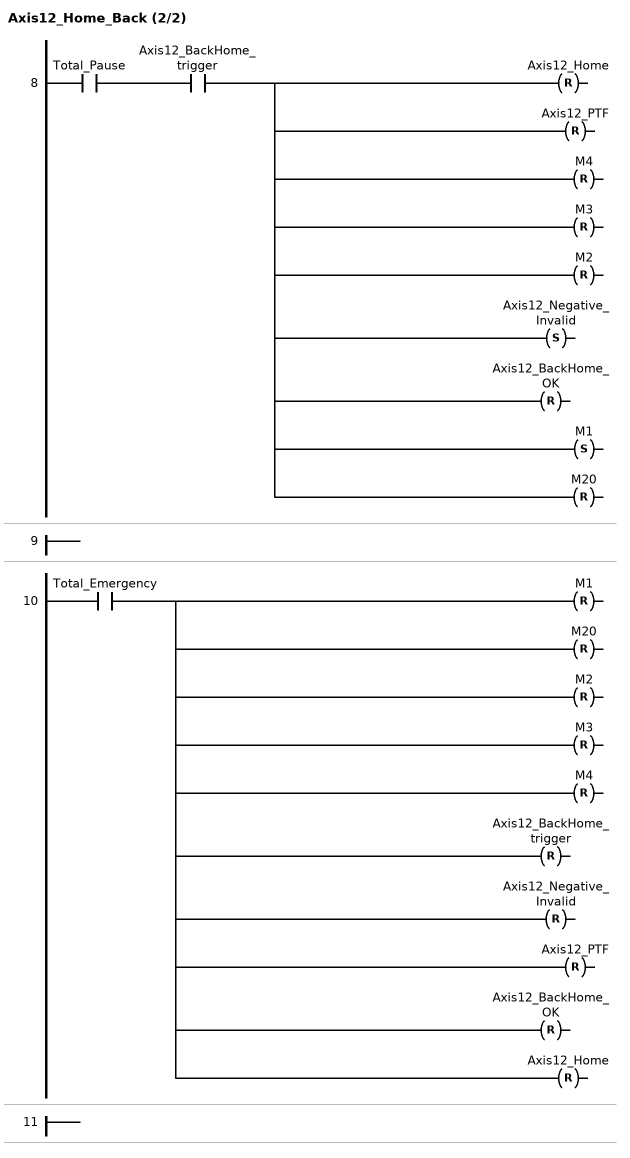
[picture p96: Axis12_Home_Back (LD)]
_LD_ (* Ladder Diagram *)
NETWORK 1
	[Axis12_BackHome_trigger] - UP1:R_TRIG(CLK: *) --- (S M1) (S Axis12_Negative_Invalid)
NETWORK 2
	[M1] - [/Total_Pause] --- (S Axis12_PTF) (S M2) (R M1)
NETWORK 3
	[M2] - [Axis12_Negative_Limit] --- (S Axis12_Halt) (S M20) (R M2) (R Axis12_PTF)
NETWORK 4
	[M20] - [Axis12_Halt_Function.Done] - T1:TON(IN: *, PT: T#1MS) --- (R Axis12_Halt) (S M3) (R M20)
NETWORK 5
	[M3] - [/Total_Pause] --- (S M4) (S Axis12_Home)
NETWORK 6
	[M4] - [Axis12_Negative_Limit] - DOWN1:F_TRIG(CLK: *) --- (R Axis12_Negative_Invalid)
NETWORK 7
	[M4] - [Axis12_Home_Function.Done] --- (S Axis12_BackHome_OK) (R Axis12_Home) (R Axis12_BackHome_trigger) (R M4) (R M3)
NETWORK 8
	[Total_Pause] - [Axis12_BackHome_trigger] --- (R Axis12_Home) (R Axis12_PTF) (R M4) (R M3) (R M2) (S Axis12_Negative_Invalid) (R Axis12_BackHome_OK) (S M1) (R M20)
NETWORK 9
	*
NETWORK 10
	[Total_Emergency] --- (R M1) (R M20) (R M2) (R M3) (R M4) (R Axis12_BackHome_trigger) (R Axis12_Negative_Invalid) (R Axis12_PTF) (R Axis12_BackHome_OK) (R Axis12_Home)
NETWORK 11
	*
_END_LD_
(* the same logic as Structured Text *)
(* Network 1 *)
UP1(CLK := Axis12_BackHome_trigger);
IF UP1.Q THEN M1 := TRUE; Axis12_Negative_Invalid := TRUE; END_IF;
(* Network 2 *)
_p1 := M1 AND NOT Total_Pause;
IF _p1 THEN Axis12_PTF := TRUE; M2 := TRUE; M1 := FALSE; END_IF;
(* Network 3 *)
_p2 := M2 AND Axis12_Negative_Limit;
IF _p2 THEN Axis12_Halt := TRUE; M20 := TRUE; M2 := FALSE; Axis12_PTF := FALSE; END_IF;
(* Network 4 *)
T1(IN := M20 AND Axis12_Halt_Function.Done, PT := T#1MS);
IF T1.Q THEN Axis12_Halt := FALSE; M3 := TRUE; M20 := FALSE; END_IF;
(* Network 5 *)
IF M3 AND NOT Total_Pause THEN M4 := TRUE; Axis12_Home := TRUE; END_IF;
(* Network 6 *)
DOWN1(CLK := M4 AND Axis12_Negative_Limit);
IF DOWN1.Q THEN Axis12_Negative_Invalid := FALSE; END_IF;
(* Network 7 *)
_p3 := M4 AND Axis12_Home_Function.Done;
IF _p3 THEN Axis12_BackHome_OK := TRUE; Axis12_Home := FALSE; Axis12_BackHome_trigger := FALSE; M4 := FALSE; M3 := FALSE; END_IF;
(* Network 8 *)
IF Total_Pause AND Axis12_BackHome_trigger THEN Axis12_Home := FALSE; Axis12_PTF := FALSE; M4 := FALSE; M3 := FALSE; M2 := FALSE; Axis12_Negative_Invalid := TRUE; Axis12_BackHome_OK := FALSE; M1 := TRUE; M20 := FALSE; END_IF;
(* Network 9 *)
(* Network 10 *)
IF Total_Emergency THEN M1 := FALSE; M20 := FALSE; M2 := FALSE; M3 := FALSE; M4 := FALSE; Axis12_BackHome_trigger := FALSE; Axis12_Negative_Invalid := FALSE; Axis12_PTF := FALSE; Axis12_BackHome_OK := FALSE; Axis12_Home := FALSE; END_IF;
(* Network 11 *)
END_PROGRAM

(* POU Other_Folder/Akam_Stop_Message/Initialization_Folder/IniRun, ST *)
PROGRAM IniRun
VAR
	step: INT;
	bak_step:INT;
	rt_hold: R_TRIG;
	M1: BOOL;

	T1: TON;
	T2:TON;


END_VAR

VAR_INPUT
	bstart1: BOOL;
	bhold1: BOOL;
	breset1: BOOL;

END_VAR
(*数据保存*)
IF Save_Button THEN
Save_Par(NETID:='',port:=801,start:=TRUE,tmout:=T#1s);
END_IF
IF NOT Save_Par.BUSY  THEN
Save_Button:=FALSE;
Save_Par(NETID:='',port:=801,start:=FALSE,tmout:=T#1s);
END_IF


(*当出现回原点没有时，需要初始化*)
IF NOT Axis1_BackHome_OK OR NOT  Axis2_BackHome_OK OR NOT Axis3_BackHome_OK OR NOT Axis4_BackHome_OK OR NOT Axis5_BackHome_OK
	OR NOT Axis6_BackHome_OK OR NOT Axis7_BackHome_OK OR NOT Axis8_BackHome_OK OR NOT Axis9_BackHome_OK OR NOT Axis10_BackHome_OK OR NOT Axis11_BackHome_OK  THEN
;(*判断是否需要回原点----------------------------------------------------*)
END_IF
(*---------------------------------------------------------------------------初始化开始流程---------------------------------------------------------------------------------*)
CASE step OF
0:
Need_Ini:=TRUE;(*此时寻妖初始化*)
(*进入初始化流程*)
step:=10;

10:(*判断是否需要初始化*)
IF Need_Ini AND NOT Total_Axis_Error AND NOT Debug_Model   THEN (*当需要初始化的时候，复位所有原点ok信号*)
	Axis1_BackHome_OK:=FALSE;
Axis2_BackHome_OK:=FALSE;
Axis3_BackHome_OK:=FALSE;
Axis4_BackHome_OK:=FALSE;
Axis5_BackHome_OK:=FALSE;
Axis6_BackHome_OK:=FALSE;
Axis7_BackHome_OK:=FALSE;
Axis8_BackHome_OK:=FALSE;
Axis9_BackHome_OK:=FALSE;
Axis10_BackHome_OK:=FALSE;
Axis11_BackHome_OK:=FALSE;
step:=20;
END_IF

20:(*等待复位按钮操作，复位报警等状态*)
IF X4_6 AND Need_Ini THEN
	IF Total_Axis_Error THEN
	M1:=TRUE;(*no use*)(*上位机提示电机报警问题，需要初始化*)
	END_IF
	IF NOT Total_Axis_Error THEN
	step:=30;
	END_IF
END_IF;

30:(*启动按下的处理开始进入初始化过中。。。。。。*)
IF X4_4 AND NOT Total_Axis_Error AND NOT Debug_Model THEN
Need_Ini:=FALSE;
IsIniing:=TRUE;(*初始化中ing*)
M101:=TRUE;(*初始化中，速度为中速*)
Axis1_Poweron:=TRUE;
Axis2_Poweron:=TRUE;
Axis3_Poweron:=TRUE;
Axis4_Poweron:=TRUE;
Axis5_Poweron:=TRUE;
Axis6_Poweron:=TRUE;
Axis7_Poweron:=TRUE;
Axis8_Poweron:=TRUE;
Axis9_Poweron:=TRUE;
Axis10_Poweron:=TRUE;
Axis11_Poweron:=TRUE;
step:=39;
END_IF

39:
(*滑台气缸上下，如果在同一高度，则说明不存在重叠部分，可复位气缸*)
IF (X4_11 AND X4_13) OR (X4_12 AND X4_14)  AND X2_6 THEN
Y1_6:=FALSE;
Y1_7:=FALSE;
step:=40;
ELSE
step:=40;
END_IF


40:(*气缸复位状态保留*)

Y0_2:=FALSE;
Y0_5:=FALSE;
Y0_14:=FALSE;
y0_1:=TRUE;
Y0_12:=FALSE;



(******************** AND  *****************************)

Y0_7:=FALSE;(*左上下气缸*)
Y0_9:=FALSE;(*滚压气缸复位*)
Y1_1:=FALSE;(*右上下气缸*)
Y0_4:=FALSE;
Y1_3:=FALSE;
IF X2_13 AND X3_3 AND X3_11 THEN
	step:=50;(*初步气缸复位*)
END_IF

50:
Y0_6:=FALSE;(*左平移气缸复位*)
Y0_11:=FALSE;(*滚压部分下压气缸复位*)
Y0_16:=FALSE;(*右平移气缸复位*)
T1(IN:=TRUE , PT:=t#1s , Q=> , ET=> );
IF T1.Q AND X2_11 AND X3_9 THEN
T1(IN:=FALSE , PT:=t#1s , Q=> , ET=> );
step:=60;(*无感气缸*)
END_IF

60:(*复位滚压气缸部分气缸，推入气缸，和翻转气缸*)
Y0_10:=FALSE;
IF X3_1 THEN
step:=70;
END_IF

70:(*翻转气缸复位*)
Y0_13:=FALSE;
IF X3_5 THEN
step:=80;
END_IF

80:(*上电延时*)
T2(IN:=TRUE , PT:=t#1s , Q=> , ET=> );
IF T2.Q  AND NOT Total_Pause THEN
T2(IN:=FALSE , PT:=t#1s , Q=> , ET=> );
step:=90;
END_IF

90:
home_backing:=TRUE;
IF NOT Axis3_BackHome_OK OR NOT Axis6_BackHome_OK OR NOT Axis7_BackHome_OK OR NOT Axis8_BackHome_OK OR NOT Axis9_BackHome_OK THEN
step:=100;
ELSE
step:=110;(*当喂料都已经回过原点，则不需要回原点*)
END_IF


100:(*判断是否都需要回原点*)(*喂料部分回原点*)
Axis3_BackHome_trigger:=TRUE;(**)
Axis6_BackHome_trigger:=TRUE;(**)
Axis7_BackHome_trigger:=TRUE;(**)
Axis8_BackHome_trigger:=TRUE;(**)
Axis9_BackHome_trigger:=TRUE;
IF Axis3_BackHome_OK AND Axis6_BackHome_OK AND Axis7_BackHome_OK AND Axis8_BackHome_OK AND Axis9_BackHome_OK  THEN
Axis3_BackHome_trigger:=FALSE;(**)
Axis6_BackHome_trigger:=FALSE;(**)
Axis7_BackHome_trigger:=FALSE;(**)
Axis8_BackHome_trigger:=FALSE;(**)
Axis9_BackHome_trigger:=FALSE;
step:=101;
END_IF

101:(*升降回到初始位置*)
D3:=D300;(*进料初始位置，在下面*)
D6:=D600;(*上升初始位置，在下面*)
D7:=D700;(*下降初始位置，在下面*)
D8:=D800;(*上升初始位置，在下面*)
D9:=D900;(*下降初始位置，在下面*)
Axis3_MoveAbsolute:=TRUE;
Axis6_MoveAbsolute:=TRUE;
Axis7_MoveAbsolute:=TRUE;
Axis8_MoveAbsolute:=TRUE;
Axis9_MoveAbsolute:=TRUE;
IF Axis3_Abs_Function.Done AND Axis6_Abs_Function.Done AND Axis7_Abs_Function.Done AND Axis8_Abs_Function.Done AND Axis9_Abs_Function.Done  THEN
Axis3_MoveAbsolute:=FALSE;
Axis6_MoveAbsolute:=FALSE;
Axis7_MoveAbsolute:=FALSE;
Axis8_MoveAbsolute:=FALSE;
Axis9_MoveAbsolute:=FALSE;
step:=102;  (*初始都在下面*)
END_IF

102:(*Z轴撕膜电机回原*)
Axis5_BackHome_trigger:=TRUE;
IF Axis5_BackHome_OK THEN
Axis5_BackHome_trigger:=FALSE;
step:=103;
END_IF

103:
D5:=A5_W0;(*Z轴回到初始位置*)
Axis5_MoveAbsolute:=TRUE;
IF Axis5_Abs_Function.Done THEN
Axis5_MoveAbsolute:=FALSE;
step:=110;
END_IF

110:(*其余轴回原点*)
Axis1_BackHome_trigger:=TRUE;
Axis11_BackHome_trigger:=TRUE;
Axis2_BackHome_trigger:=TRUE;
Axis4_BackHome_trigger:=TRUE;
Axis10_BackHome_trigger:=TRUE;
IF Axis1_BackHome_OK AND Axis2_BackHome_OK AND Axis4_BackHome_OK  AND Axis10_BackHome_OK AND Axis11_BackHome_OK  THEN
Axis1_BackHome_trigger:=FALSE;
Axis2_BackHome_trigger:=FALSE;
Axis4_BackHome_trigger:=FALSE;
Axis10_BackHome_trigger:=FALSE;
Axis11_BackHome_trigger:=FALSE;
step:=120;
END_IF

120:(*移载等轴的回到初始位置*)
D1:=A1_W0;
D1_1:=A11_W0+250;(*为了保证回原点之后，滑台1气缸在下面，滑台2气缸在上面，则需要，错开初始位置*)
D2:=A2_W0;
D4:=A4_W0;
D10:=A10_W0;
Axis1_MoveAbsolute:=TRUE;
Axis2_MoveAbsolute:=TRUE;
Axis4_MoveAbsolute:=TRUE;
Axis10_MoveAbsolute:=TRUE;
Axis11_MoveAbsolute:=TRUE;
IF Axis1_Abs_Function.Done AND Axis2_Abs_Function.Done AND Axis4_Abs_Function.Done  AND Axis10_Abs_Function.Done AND Axis11_Abs_Function.Done  THEN
Axis1_MoveAbsolute:=FALSE;
Axis2_MoveAbsolute:=FALSE;
Axis4_MoveAbsolute:=FALSE;
Axis10_MoveAbsolute:=FALSE;
Axis11_MoveAbsolute:=FALSE;
home_backing:=FALSE;
Y1_6:=FALSE;(*最终保证，滑台1在上面，滑台2气缸在下面*)
Y1_7:=FALSE;
step:=121;
END_IF


121:
IF  X4_11 AND X4_14 THEN(*最终结果，传感器检测*)
step:=122;
END_IF

122:
D1_1:=A11_W0;
Axis11_MoveAbsolute:=TRUE;
IF  Axis11_Abs_Function.Done THEN
Axis11_MoveAbsolute:=FALSE;
step:=130;
END_IF


130:(*其余需要初始化的状态*)

IsIniing:=FALSE;
Model_Choose:=TRUE;(*模式选择*)
step:=140;

140:
(*模式选选择，直接按钮，启动程序，当选上位机选择调试模式，同时按下启动按钮，则进入调试模式*)
IF NOT Debug_Model AND X4_4 THEN
	Model_Choose:=FALSE;(*模式选择*)
Product_Film_Handel_Run:=TRUE;
Left_Translation_Run_1:=TRUE;
Left_Translation_Run_2:=TRUE;
Right_Translation_Run:=TRUE;
Rolling_Part_Run:=TRUE;
Right_Carry_Run:=TRUE;
Left_Carry_Run:=TRUE;
Liftin_Feed_1_Run:=TRUE;
Liftin_Feed_Left_1_Run:=TRUE;
Liftin_Feed_Left_2_Run:=TRUE;
Liftin_Feed_Right_1_Run:=TRUE;
Liftin_Feed_Right_2_Run:=TRUE;
M102:=TRUE;
Debug_Model:=FALSE;
Positive2_Safe:=TRUE;
	Positive3_Safe:=TRUE;
	Positive_Wait_Safe:=TRUE;
runing:=TRUE;
	step:=150;
END_IF
IF Debug_Model AND X4_4 THEN
	M100:=TRUE;(*调试模式下低速*)
	Model_Choose:=FALSE;(*模式选择*)
	Axis1_debug_trigger:=TRUE;
Axis1_debug_trigger:=TRUE;
Axis2_debug_trigger:=TRUE;
Axis3_debug_trigger:=TRUE;
Axis4_debug_trigger:=TRUE;
Axis5_debug_trigger:=TRUE;
Axis6_debug_trigger:=TRUE;
Axis7_debug_trigger:=TRUE;
Axis8_debug_trigger:=TRUE;
Axis9_debug_trigger:=TRUE;
Axis10_debug_trigger:=TRUE;
Axis11_debug_trigger:=TRUE;
(*其余调试模式*)
 step:=160;
END_IF

150:(*运行模式下的死循环*)
;


160:
(*调试模式下的死循环，等待调试模式借宿，重新开始初始化*)
IF NOT Debug_Model THEN
Need_Ini:=TRUE;
 	    bak_step:=0;
	step:=0;
END_IF



300:(*外部输入启动*)
    IF bstart1   AND NOT Total_Axis_Error AND NOT total_pausestatus THEN
	step:=bak_step;
END_IF;
END_CASE;



(*触发暂停的外部输入*)
rt_hold(CLK:=( Total_Axis_Error OR  bhold1) , Q=> ); (*暂停状态*)
IF step<>0 AND step<>300   AND  rt_hold.Q THEN
     bak_step:=step;
     step:=300;
END_IF

(*急停处理*)
IF Total_Emergency THEN
debug_FLIG:=FALSE;
M100:=FALSE;
M101:=FALSE;
M102:=FALSE;
IsIniing:=FALSE;
runing:=FALSE;
home_backing:=FALSE;
Model_Choose:=FALSE;(*模式选择*)


Debug_Model:=FALSE;
Positive2_Safe:=FALSE;
Positive3_Safe:=FALSE;
Positive_Wait_Safe:=FALSE;


bak_step:=0;
step:=0;
END_IF


(*与debug1中的梯形图一起使用，当不在应该调试模式下的时候，按下调试按钮，自动复位--------详见------debug1----------*)
IF step<>160 AND step<>140 AND step<>300  THEN
debug_FLIG:=FALSE;
ELSE
debug_FLIG:=TRUE;
END_IF
END_PROGRAM

(* POU old/Old_Tray_Pro/Liftin_Feed_Right_1, ST *)
PROGRAM Liftin_Feed_Right_1
VAR

	step: INT;
	bak_step:INT;
	rt_hold: R_TRIG;
	UP1: R_TRIG;
	T1: TON;
	T2:TON;

END_VAR

VAR_INPUT
	bstart1: BOOL;
	bhold1: BOOL;
	breset1: BOOL;

END_VAR
UP1(CLK:=Liftin_Feed_Right_1_Run , Q=> );

CASE step OF
0:
 IF UP1.Q THEN
step:=10;
END_IF


10:(*上升运行*)
Axis8_PTF_2:=TRUE;
IF X2_4 AND  X1_3 THEN(*碰到光纤，同时没有碰到极限，此时上料ok*)
Axis8_PTF_2:=FALSE;
Feed_3_Finish:=TRUE;
Axis8_Halt:=TRUE;
step:=20;
END_IF
IF NOT X1_3 THEN(*碰到极限，此时表示料空*)
Axis8_PTF_2:=FALSE;
Axis8_Halt:=TRUE;
step:=50;
END_IF

20:
Axis8_Halt:=FALSE;
(*表示上料成功,等待取完信号*)
IF Get_Robort3_Tray_Full THEN
Feed_3_Finish:=FALSE;
Get_Robort3_Tray_Full:=FALSE;(*放满信号，给出，等待移动*)
Right_Can_Move:=TRUE;
step:=30;
END_IF


30:(*等待平移完成，才可以上升*)
IF Right_Move_Finish THEN
Right_Move_Finish:=FALSE;
step:=10;
END_IF


50:(*碰到极限，此时料取完,回到初始位置*)
Axis8_Halt:=FALSE;
D8:=D800;
Axis8_MoveAbsolute:=TRUE;
IF Axis8_Abs_Function.Done THEN
Axis8_MoveAbsolute:=FALSE;
Feed_Right_None_Alam:=TRUE;(*不暂停，只提示*)
step:=60;
END_IF

60:(*回到初始位置，提示料空*)
IF Right_UP_Button AND NOT Total_Pause THEN
Right_UP_Button:=FALSE;
Feed_Right_None_Alam:=FALSE;(*不暂停，只提示*)
step:=10;
END_IF

300:
    IF bstart1   AND NOT Total_Axis_Error AND NOT total_pausestatus THEN
	step:=bak_step;
END_IF;
END_CASE


rt_hold(CLK:=( Total_Axis_Error OR  bhold1) , Q=> ); (*暂停状态*)
IF step<>0 AND step<>300   AND  rt_hold.Q THEN
     bak_step:=step;
     step:=300;
END_IF


IF Right_UP_Button THEN
Right_UP_Button:=FALSE;
END_IF

IF Total_Emergency THEN
Liftin_Feed_Right_1_Run:=FALSE;
Feed_Right_None_Alam:=FALSE;
Feed_3_Finish:=FALSE;


bak_step:=0;
step:=0;
END_IF


(*随时可以不做料的操作*)
IF Feed_Right_Button1 AND step=20 AND NOT Total_Pause THEN
Feed_Right_Button1:=FALSE;
Feed_3_Finish:=FALSE;
step:=50;
ELSE
Feed_Right_Button1:=FALSE;
END_IF
END_PROGRAM

(* POU old/Old_Tray_Pro/Liftin_Feed_Right_2, ST *)
PROGRAM Liftin_Feed_Right_2
VAR

	step: INT;
	bak_step:INT;
	rt_hold: R_TRIG;
	UP1: R_TRIG;
	DOWN1: F_TRIG;

	T1: TON;
	T2:TON;

END_VAR

VAR_INPUT
	bstart1: BOOL;
	bhold1: BOOL;
	breset1: BOOL;

END_VAR
(*左下降，初始化，回原点到初始位置，，，启动之后，先往上走，到初始位置(第一次回原点使用)  ，接收到送料完成可下降信号，则
开始下降，等现将结束，告知，可放料*)

UP1(CLK:=Liftin_Feed_Right_2_Run , Q=> );

CASE step OF
0:
 IF UP1.Q THEN
step:=1;
END_IF

1:
(*初始化之后位置在下面的初始位置*)
Axis9_PTF_2:=TRUE;
IF X2_5 AND X1_6 THEN
Axis9_PTF_2:=FALSE;
Axis9_Halt:=TRUE;
step:=20;
END_IF
IF NOT X1_6 THEN
Axis9_PTF_2:=FALSE;
Axis9_Halt:=TRUE;
step:=60;(*撞到极限，此时需要回到上面的初始位置*)
END_IF

10:
(*初始化的时候写，回原点之后，向上跑知道碰到光纤，或者极限的时候，到极限回到初始位置，碰到光纤，停止，翻转到极限停止位置*)

(*到初始位置，等待放料，当光纤感应到，同时，接收到，可下降信号的时候，开始下降，当感应不到光纤，则停止*)
IF you_ke_jiang AND X2_5 THEN
you_ke_jiang:=FALSE;
	step:=20;
END_IF

20:
Axis9_Halt:=FALSE;
(*接收到可降信号，开始下降，到传感器下降沿停止下降，等待*)
Axis9_PTF:=TRUE;
DOWN1(CLK:=X2_5 , Q=> );
IF DOWN1.Q AND NOT  X1_7 THEN
Axis9_PTF:=FALSE;
you_down_Finish:=TRUE;
Axis9_Halt:=TRUE;
step:=30;
END_IF
IF  X1_7 THEN(*碰到极限，此时表示料空*)
Axis9_PTF:=FALSE;
Axis9_Halt:=TRUE;
step:=400;
END_IF

30:(*停止，给出下降完成信号，等待放料循环*)
Axis9_Halt:=FALSE;
step:=10;

400:(*碰到原点，此时，回到下初始位置，给出料满提示*)
Axis9_Halt:=FALSE;
D9:=D900;
Axis9_MoveAbsolute:=TRUE;
IF Axis9_Abs_Function.Done THEN
Axis9_MoveAbsolute:=FALSE;
Feed_Right_None_Alam:=TRUE;(*不暂停，只提示*)
step:=50;
END_IF

50:(*碰到下极限，给出缺料提示*)
Axis9_Halt:=FALSE;
IF Right_Down_Button AND NOT Total_Pause THEN
	Right_Down_Button:=FALSE;
Feed_Right_Full_Alam:=FALSE;
	step:=1;(*确认拿走料之后，运动到初始位置*)
END_IF

60:(*回到初始位置*)
Axis9_Halt:=FALSE;
D9:=D910;
Axis9_MoveAbsolute:=TRUE;
IF Axis9_Abs_Function.Done THEN
Axis9_MoveAbsolute:=FALSE;
you_down_Finish:=TRUE;(*左下降完成信号*)
step:=10;
END_IF

300:
    IF bstart1   AND NOT Total_Axis_Error AND NOT total_pausestatus THEN
	step:=bak_step;
END_IF;
END_CASE


rt_hold(CLK:=( Total_Axis_Error OR  bhold1) , Q=> ); (*暂停状态*)
IF step<>0 AND step<>300   AND  rt_hold.Q THEN
     bak_step:=step;
     step:=300;
END_IF


IF Total_Emergency THEN
Liftin_Feed_Right_2_Run:=FALSE;
you_down_Finish:=FALSE;
Feed_Right_Full_Alam:=FALSE;


bak_step:=0;
step:=0;
END_IF


(*随时可以不做料的操作*)
IF Feed_Right_Button2 AND step=10 AND NOT Total_Pause THEN
Feed_Right_Button2:=FALSE;
you_down_Finish:=FALSE;
step:=400;
ELSE
Feed_Right_Button2:=FALSE;
END_IF
END_PROGRAM

(* POU Test_Part_pro/New_Table_3, ST *)
PROGRAM New_Table_3
VAR
	step: INT;
	bak_step:INT;
	rt_hold: R_TRIG;
	UP1: R_TRIG;
	Run_Time:BOOL;
	T1:TON;
	Run_Time_Lreal: TIME;




	T2: TON;
	T3: TON;
END_VAR

VAR_INPUT
	bstart1: BOOL;
	bhold1: BOOL;
	breset1: BOOL;

END_VAR
UP1(CLK:=Left_Translation_Run_2 , Q=> );

CASE step OF
0:
 IF UP1.Q THEN
step:=10;
END_IF

10:
D1_1:=A11_W1;(*左等待放料工位*)
Axis11_MoveAbsolute:=TRUE;
IF Axis11_Abs_Function.Done THEN
Axis11_MoveAbsolute:=FALSE;
step:=20;
END_IF;

20:(*到下初始位置------寻味位置1是否安全*)
IF Positive1_Safe THEN
	Positive1_Safe:=FALSE;
	Y1_7:=TRUE;
step:=30;
END_IF

30:
IF X4_13 THEN
	Positive4_Safe:=TRUE;
	step:=40;
END_IF

40:(*安全之后上顶*)
IF Tray2_Have THEN
	step:=72;
ELSE
step:=72;
END_IF

50:(*到位置之后，告知可以放料*)
D1_1:=A11_W1;(*左等待放料工位*)
Axis11_MoveAbsolute:=TRUE;
IF Axis11_Abs_Function.Done THEN
Process_2_Can_Push:=TRUE;
Axis11_MoveAbsolute:=FALSE;
Y0_2:=TRUE;
step:=60;
END_IF;

60:(*上料-----等待放下之后---------*)
IF Process_1_Push_Finish THEN
Tray2_Have:=TRUE;
Process_1_Push_Finish:=FALSE;
step:=70;
END_IF

70:
T2(IN:=TRUE , PT:=t#1s , Q=> , ET=> );
   IF T2.Q AND NOT Total_Pause  THEN
T2(IN:=FALSE, PT:=t#1S , Q=> , ET=> );
Can_Move_Film:=TRUE;(*给出可撕膜信号*)
step:=71;
END_IF

71:(*撕膜完成信号等到*)
IF Process_1_Push_Finish_Sure THEN
Process_1_Push_Finish_Sure:=FALSE;
step:=72;
END_IF

72:(*判断拍照位置1是否安全*)
IF Positive_Camera_Safe1 THEN
Positive_Camera_Safe1:=FALSE;(*拍照位置1被占据*)
step:=73;
END_IF

73:
D1_1:=A11_W2;(*拍照工位1*)
Axis11_MoveAbsolute:=TRUE;
IF Axis11_Abs_Function.Done THEN
Axis11_MoveAbsolute:=FALSE;
(*到位拍照*)
step:=90;
END_IF

80:(*拍照工位1拍照结束-----等待*)
IF Camera_1_5_OK THEN
Camera_1_5_run:=FALSE;
Camera_1_5_OK:=FALSE;
step:=90;
END_IF
IF Camera1_NG THEN  (*拍照失败的处理，判断ng,此时需要给出结果，，，，，，，同时运动到工作位置*)
Camera_1_5_run:=FALSE;
Tray2_Have:=FALSE;
Camera1_NG:=FALSE;
Y0_2:=FALSE;
step:=2000;
END_IF

90:(*判断拍照位置2是否安全*)
IF Positive_Camera_Safe2 THEN
Positive_Camera_Safe2:=FALSE;
step:=100;
END_IF

100:(*移动到位置2*)
D1_1:=A11_W3; (*拍照工位2*)
Axis11_MoveAbsolute:=TRUE;
IF Axis11_Abs_Function.Done THEN
Axis11_MoveAbsolute:=FALSE;
(*到位拍照*)
step:=120;
END_IF

110:
IF Camera_1_6_OK THEN
Camera_1_6_run:=FALSE;
Camera_1_6_OK:=FALSE;
step:=120;
END_IF
IF Camera1_NG THEN  (*拍照失败的处理，判断ng,此时需要给出结果，，，，，，，同时运动到工作位置*)
Camera_1_6_run:=FALSE;
Tray2_Have:=FALSE;
Camera1_NG:=FALSE;
Y0_2:=FALSE;
step:=2020;
END_IF


120:(*判断位置3是否安全*)
IF Positive_Camera_Safe3 THEN
Positive_Camera_Safe3:=FALSE;
step:=130;
END_IF

130:(*到工位3*)
D1_1:=A11_W4;(*拍照工位3*)
Axis11_MoveAbsolute:=TRUE;
IF Axis11_Abs_Function.Done THEN
Axis11_MoveAbsolute:=FALSE;
(*到位拍照*)
step:=150;
END_IF

140:
IF Camera_1_7_OK THEN
Camera_1_7_run:=FALSE;
Camera_1_7_OK:=FALSE;
step:=150;
END_IF
IF Camera1_NG THEN  (*拍照失败的处理，判断ng,此时需要给出结果，，，，，，，同时运动到工作位置*)
Camera_1_7_run:=FALSE;
Tray2_Have:=FALSE;
Camera1_NG:=FALSE;
Y0_2:=FALSE;
step:=2050;
END_IF

150:(*拍照位置3判断是否安全----------*)
IF Positive_Camera_Safe4 THEN
Positive_Camera_Safe4:=FALSE;
step:=160;
END_IF

160:
D1_1:=A11_W5;(*拍照工位4*)
Axis11_MoveAbsolute:=TRUE;
IF Axis11_Abs_Function.Done THEN
Axis11_MoveAbsolute:=FALSE;
(*到位拍照*)

Positive1_Safe:=TRUE;
step:=180;
END_IF

170:
IF Camera_1_8_OK THEN
Camera_1_8_run:=FALSE;
Camera_1_8_OK:=FALSE;
step:=180;
END_IF
IF Camera1_NG THEN  (*拍照失败的处理，判断ng,此时需要给出结果，，，，，，，同时运动到工作位置*)
Camera_1_8_run:=FALSE;
Tray2_Have:=FALSE;
Camera1_NG:=FALSE;
Y0_2:=FALSE;
step:=2070;
END_IF

180:(*判断工作位置1是否安全*)
IF Positive_Fit_Safe1 THEN
Positive_Fit_Safe1:=FALSE;
(*
HB_Fit_Finish_5:=FALSE;
HB_Fit_Finish_6:=FALSE;
HB_Fit_Finish_7:=FALSE;
HB_Fit_Finish_8:=FALSE;*)
step:=190;
END_IF

190:(*到工作位置1*)
D1_1:=A11_W6;(*工作位置工位1*)
Axis11_MoveAbsolute:=TRUE;
IF Axis11_Abs_Function.Done THEN
Axis11_MoveAbsolute:=FALSE;

Positive_Camera_Safe1:=TRUE;(*工作位置1是给出拍照位置1安全安全位置-------------------------------------*)

step:=210;
END_IF

200:(*到位等待贴合完成*)
IF HB_Fit_Finish_5 THEN
FG_Ready_5:=FALSE;
HB_Fit_Finish_5:=FALSE;
step:=210;
END_IF

210:(*工位1贴合完成-----询问工作位置2是否安全*)
IF Positive_Fit_Safe2 THEN
Positive_Fit_Safe2:=FALSE;
step:=220;
END_IF

220:(*位置安全------到贴合位置2*)
D1_1:=A11_W7;(*工作位置工位1*)
Axis11_MoveAbsolute:=TRUE;
IF Axis11_Abs_Function.Done THEN
Axis11_MoveAbsolute:=FALSE;

Positive_Camera_Safe2:=TRUE;(*工作位置1是给出拍照位置1安全安全位置-------------------------------------*)

step:=240;
END_IF

230:(*等待贴合完成信号*)
IF HB_Fit_Finish_6 THEN
FG_Ready_6:=FALSE;
HB_Fit_Finish_6:=FALSE;
step:=240;
END_IF

240:(*贴合完成------寻问位置3是否安全*)
IF Positive_Fit_Safe3 THEN
Positive_Fit_Safe3:=FALSE;
step:=250;
END_IF

250:(*位置安全------到贴合位置2*)
D1_1:=A11_W8;(*工作位置工位1*)
Axis11_MoveAbsolute:=TRUE;
IF Axis11_Abs_Function.Done THEN
Axis11_MoveAbsolute:=FALSE;

Positive_Camera_Safe3:=TRUE;(*工作位置1是给出拍照位置1安全安全位置-------------------------------------*)

step:=270;
END_IF

260:(*等待贴合完成信号*)
IF HB_Fit_Finish_7 THEN
FG_Ready_7:=FALSE;
HB_Fit_Finish_7:=FALSE;
step:=270;
END_IF

270:(*位置3贴合完成，询问位置4是否安全*)
IF Positive_Fit_Safe4 THEN
Positive_Fit_Safe4:=FALSE;
step:=280;
END_IF

280:(*位置安全------到贴合位置2*)
D1_1:=A11_W9;(*工作位置工位1*)
Axis11_MoveAbsolute:=TRUE;
IF Axis11_Abs_Function.Done THEN
Axis11_MoveAbsolute:=FALSE;

Positive_Camera_Safe4:=TRUE;(*工作位置1是给出拍照位置1安全安全位置-------------------------------------*)

step:=300;
END_IF

290:(*等待贴合完成信号*)
IF HB_Fit_Finish_8 THEN
FG_Ready_8:=FALSE;
HB_Fit_Finish_8:=FALSE;
step:=300;
END_IF

300:
IF Positive2_Safe THEN
	Positive2_Safe:=FALSE;
	step:=350;
END_IF

310:(*位置到位后，等待，送吸嘴*)
IF Wait_Robort2_Touch_Finish  THEN
Wait_Robort2_Touch_Finish:=FALSE;
Y0_2:=FALSE;
step:=320;
END_IF

320:
T3(IN:=TRUE , PT:=t#1s , Q=> , ET=> );
   IF T3.Q AND NOT Total_Pause  THEN
T3(IN:=FALSE, PT:=t#1S , Q=> , ET=> );
step:=340;
END_IF

340:
IF Get_Robot1_Get_Finish THEN
Tray2_Have:=FALSE;
Get_Robot1_Get_Finish:=FALSE;
step:=350;
END_IF

350:
IF Positive3_Safe THEN
	Positive3_Safe:=FALSE;
	Y1_7:=FALSE;
	step:=360;
END_IF

360:
IF X4_14 THEN
Positive2_Safe:=TRUE;
Positive_Fit_Safe1:=TRUE;
Positive_Fit_Safe2:=TRUE;
Positive_Fit_Safe3:=TRUE;
Positive_Fit_Safe4:=TRUE;

	step:=370;
END_IF

370:(*下降之后，*)
IF Positive4_Safe THEN
	Positive4_Safe:=FALSE;
	step:=380;
END_IF

380:
D1_1:=A11_W1;(*左等待放料工位------下的位置*)
Axis11_MoveAbsolute:=TRUE;
IF Axis11_Abs_Function.Done THEN
Axis11_MoveAbsolute:=FALSE;
Positive3_Safe:=TRUE;
step:=10;
END_IF;



600:
    IF bstart1   AND NOT Total_Axis_Error  AND NOT total_pausestatus THEN
	step:=bak_step;
END_IF;



2000:(*拍照位置1NG------------处理*)
IF Positive_Camera_Safe2 THEN
Positive_Camera_Safe2:=FALSE;
step:=2010;
END_IF

2010:(*移动到位置2*)
D1_1:=A11_W3; (*拍照工位2*)
Axis11_MoveAbsolute:=TRUE;
IF Axis11_Abs_Function.Done THEN
Axis11_MoveAbsolute:=FALSE;
(*到位拍照*)
step:=2020;
END_IF

2020:(*拍照位置2------ng处理*)
IF Positive_Camera_Safe3 THEN
Positive_Camera_Safe3:=FALSE;
step:=2040;
END_IF

2040:(*移动到位置2*)
D1_1:=A11_W4; (*拍照工位3*)
Axis11_MoveAbsolute:=TRUE;
IF Axis11_Abs_Function.Done THEN
Axis11_MoveAbsolute:=FALSE;
(*到位拍照*)
step:=2050;
END_IF

2050:(*拍照位置2------ng处理*)
IF Positive_Camera_Safe4 THEN
Positive_Camera_Safe4:=FALSE;
step:=2060;
END_IF

2060:(*移动到位置2*)
D1_1:=A11_W5; (*拍照工位3*)
Axis11_MoveAbsolute:=TRUE;
IF Axis11_Abs_Function.Done THEN
Axis11_MoveAbsolute:=FALSE;
Positive1_Safe:=TRUE;
(*到位拍照*)
step:=2070;
END_IF


2070:(*拍照*)
IF Positive_Fit_Safe1 THEN
Positive_Fit_Safe1:=FALSE;
step:=2080;
END_IF

2080:(*到工作位置1*)
D1_1:=A11_W6;(*工作位置工位1*)
Axis11_MoveAbsolute:=TRUE;
IF Axis11_Abs_Function.Done THEN
Positive_Camera_Safe1:=TRUE;(*工作位置1是给出拍照位置1安全安全位置-------------------------------------*)
Axis11_MoveAbsolute:=FALSE;
step:=2090;
END_IF

2090:(*拍照*)
IF Positive_Fit_Safe2 THEN
Positive_Fit_Safe2:=FALSE;
step:=2100;
END_IF

2100:(*到工作位置1*)
D1_1:=A11_W7;(*工作位置工位1*)
Axis11_MoveAbsolute:=TRUE;
IF Axis11_Abs_Function.Done THEN
Positive_Camera_Safe2:=TRUE;(*工作位置1是给出拍照位置1安全安全位置-------------------------------------*)
Axis11_MoveAbsolute:=FALSE;
step:=2110;
END_IF

2110:
IF Positive_Fit_Safe3 THEN
Positive_Fit_Safe3:=FALSE;
step:=2120;
END_IF

2120:(*到工作位置1*)
D1_1:=A11_W8;(*工作位置工位1*)
Axis11_MoveAbsolute:=TRUE;
IF Axis11_Abs_Function.Done THEN
Positive_Camera_Safe3:=TRUE;(*工作位置1是给出拍照位置1安全安全位置-------------------------------------*)
Axis11_MoveAbsolute:=FALSE;
step:=2130;
END_IF

2130:
IF Positive_Fit_Safe4 THEN
Positive_Fit_Safe4:=FALSE;
step:=2140;
END_IF

2140:(*到工作位置1*)
D1_1:=A11_W9;(*工作位置工位1*)
Axis11_MoveAbsolute:=TRUE;
IF Axis11_Abs_Function.Done THEN
Positive_Camera_Safe4:=TRUE;(*工作位置1是给出拍照位置1安全安全位置-------------------------------------*)
Axis11_MoveAbsolute:=FALSE;
step:=2150;
END_IF

2150:(*贴合位置4状态此时询问位置2是否安全*)
IF Positive2_Safe THEN
	Positive2_Safe:=FALSE;
	step:=350;(*此位置寻味位置3是否安全-------------跳转*)
END_IF



END_CASE



rt_hold(CLK:=( Total_Axis_Error OR  bhold1) , Q=> ); (*暂停状态*)
IF step<>0 AND step<>600   AND  rt_hold.Q THEN
     bak_step:=step;
     step:=600;
END_IF

IF Total_Emergency THEN
Left_Translation_Run_2:=FALSE;
Process_2_Can_Push:=FALSE;(*告知上料部分可以上料*)
Can_Move_Film:=FALSE;
Tray2_Have:=FALSE;

Camera_1_5_run:=FALSE;
Camera_1_6_run:=FALSE;
Camera_1_7_run:=FALSE;
Camera_1_8_run:=FALSE;
Positive1_Safe:=FALSE;
Positive2_Safe:=FALSE;
Positive3_Safe:=FALSE;
Positive4_Safe:=FALSE;
Camera_1_5_OK:=FALSE;
Camera_1_6_OK:=FALSE;
Camera_1_7_OK:=FALSE;
Camera_1_8_OK:=FALSE;

Positive_Fit_Safe1:=FALSE;
Positive_Fit_Safe2:=FALSE;
Positive_Fit_Safe3:=FALSE;
Positive_Fit_Safe4:=FALSE;
FG_Ready_5:=FALSE;
FG_Ready_6:=FALSE;
FG_Ready_7:=FALSE;
FG_Ready_8:=FALSE;
HB_Fit_Finish_5:=FALSE;
HB_Fit_Finish_6:=FALSE;
HB_Fit_Finish_7:=FALSE;
HB_Fit_Finish_8:=FALSE;
Wait_Robort2_Touch_Finish:=FALSE;
Get_Robot1_Get_Finish:=FALSE;
Process_2_Set_Finish2:=FALSE;(*给机械手可贴合信号*)



bak_step:=0;
step:=0;
END_IF
END_PROGRAM

(* POU old/Old_Tray_Pro/Right_Carry, ST *)
PROGRAM Right_Carry
VAR
	step: INT;
	bak_step:INT;
	rt_hold: R_TRIG;
	UP1: R_TRIG;
	T1: TON;

	T2: TON;

END_VAR

VAR_INPUT
	bstart1: BOOL;
	bhold1: BOOL;
	breset1: BOOL;

END_VAR
UP1(CLK:=Right_Carry_Run , Q=> );

CASE step OF
0:
 IF UP1.Q THEN
step:=10;
END_IF

(*等待机械手取完信号，当移载完成之后，给左可上升信号，放下料之后给出，左可下降信号*)
10:
IF Right_hand_have THEN
(*手上有料，则直接放料位置*)
step:=80;
ELSE
step:=20;
END_IF

20:(*判断是否机械手取空*)
IF Right_Can_Move THEN
Right_Can_Move:=FALSE;
step:=30;
Y0_16:=TRUE;(*推杆气缸侗族*)
END_IF

30:
IF X3_8 THEN
Y1_1:=TRUE;
step:=40;
END_IF

40:
IF X3_10 THEN
Y1_2:=TRUE;
step:=50;
END_IF

50:
T1(IN:=TRUE , PT:=t#0.8s , Q=> , ET=> );
   IF T1.Q AND NOT Total_Pause  THEN
T1(IN:=FALSE, PT:=t#0.8S , Q=> , ET=> );
Y1_1:=FALSE;
step:=60;
END_IF

60:
IF X3_11 THEN(*气缸上抬到位*)
step:=70;
END_IF

70:(*判断是否吸取成功*)
IF X3_12 THEN
Y0_16:=FALSE;
step:=80;
(*吸取成功*)
ELSE
step:=30;(*重复吸取-----等待成功*)
Pressure_Right_Fail:=TRUE;
END_IF

80:(*成功之后----给出可以上顶*)
IF X3_9 THEN
Right_Move_Finish:=TRUE;
step:=90;
END_IF

90:(*上方询问是否可放*)
IF you_down_Finish THEN
you_down_Finish:=FALSE;
Y1_1:=TRUE;
step:=100;
END_IF

100:
IF X3_10 THEN
Y1_2:=FALSE;
step:=110;
END_IF

110:
T2(IN:=TRUE , PT:=t#0.8s , Q=> , ET=> );
   IF T2.Q AND NOT Total_Pause  THEN
T2(IN:=FALSE, PT:=t#0.8S , Q=> , ET=> );
Y1_1:=FALSE;
step:=120;
END_IF

120:
IF X3_11 THEN
you_ke_jiang:=TRUE;
step:=10;
END_IF

300:
    IF bstart1   AND NOT Total_Axis_Error AND NOT total_pausestatus THEN
	step:=bak_step;
END_IF;
END_CASE

rt_hold(CLK:=( Total_Axis_Error OR  bhold1) , Q=> ); (*暂停状态*)
IF step<>0 AND step<>300   AND  rt_hold.Q THEN
     bak_step:=step;
     step:=300;
END_IF

IF Total_Emergency THEN
Right_Carry_Run:=FALSE;
you_ke_jiang:=FALSE;
Right_Move_Finish:=FALSE;
bak_step:=0;
step:=0;
END_IF
END_PROGRAM

(* POU Test_Part_pro/Rolling_Part_Just, ST *)
PROGRAM Rolling_Part_Just
VAR
	step: INT;
	bak_step:INT;
	rt_hold: R_TRIG;
	UP1: R_TRIG;
	T1: TON;
	T2:TON;

	T6: TON;

	MMMM: BOOL;
	aaaa: BOOL;
END_VAR

VAR_INPUT
	bstart1: BOOL;
	bhold1: BOOL;
	breset1: BOOL;

END_VAR
UP1(CLK:=Rolling_Part_Run , Q=> );

CASE step OF
0:
 IF UP1.Q THEN
step:=10;
END_IF

10:(*滚压部分开始动作*)
(*判断机械手是否放好料---------放好之后，进行滚压动作，询问右移载是否可以送料，可送料之后，给出料，同时，发出，给料完成信号*)
step:=20;

20:(*无料的操作*)
D10:=A10_W2;
Axis10_MoveAbsolute:=TRUE;
IF Axis10_Abs_Function.Done THEN
Axis10_MoveAbsolute:=FALSE;
Process_3_Can_Push:=TRUE;
step:=29;
END_IF

29:(*机械手2放下后，告知可以开吸嘴*)
IF Wait_Robot_Push THEN
Wait_Robot_Push:=FALSE;
step:=31;
END_IF

31:
	IF Empty_Pro THEN

	step:=3000;
	ELSE
Y0_12:=TRUE;(*滚压平台*)
	step:=3000;
END_IF


3000:
IF aaaa THEN
aaaa:=FALSE;
Process_3_Set_Finish:=TRUE;
step:=10;
END_IF




30:(*等待机械手2.放料*)
IF Robot2_Push_Finish THEN
Rolling_Number:=0;
rolling_have_liao:=TRUE;
Process_3_Can_Push:=FALSE;
Robot2_Push_Finish:=FALSE;
Y0_10:=TRUE;(*推入气缸*)
step:=50;
END_IF


50:
IF X2_16 THEN
Y0_9:=TRUE;
Y0_11:=TRUE;
step:=60;
END_IF

60:
IF X3_2  THEN(*压合气缸到位，等待滚压*)
step:=70;
END_IF

70:
D10_1:=A10_W1;(*出去位置*)(*滚压低速*)
Axis10_MoveAbsolute1:=TRUE;
IF Axis10_Abs_Function1.Done THEN
Axis10_MoveAbsolute1:=FALSE;
Y0_9:=FALSE;
Y0_11:=FALSE;
step:=78;
END_IF

78:
IF X3_3 THEN
step:=80;
END_IF

80:
D10:=A10_W2;
Axis10_MoveAbsolute:=TRUE;
IF Axis10_Abs_Function.Done THEN
Axis10_MoveAbsolute:=FALSE;
Rolling_Number:=Rolling_Number+1;
step:=90;
END_IF

90:
IF Rolling_Number>=Set_Rolling_Number THEN
Rolling_Number:=0;

Y0_9:=FALSE;
step:=100;(*次数满足，跳转*)
ELSE
step:=50;
END_IF

100:
IF X3_3 THEN
Y0_10:=FALSE;
step:=110;
END_IF

110:
IF X3_1 THEN
Y0_12:=FALSE;
step:=120;
END_IF

120:
IF MMMM THEN
MMMM:=FALSE;
Process_3_Set_Finish:=TRUE;
step:=10;
END_IF



300:
    IF bstart1   AND NOT Total_Axis_Error  AND NOT total_pausestatus THEN
	step:=bak_step;
END_IF;
END_CASE

rt_hold(CLK:=( Total_Axis_Error OR  bhold1) , Q=> ); (*暂停状态*)
IF step<>0 AND step<>300   AND  rt_hold.Q THEN
     bak_step:=step;
     step:=300;
END_IF



IF Total_Emergency THEN
Rolling_Part_Run:=FALSE;
Process_3_Set_Finish:=FALSE;
Process_3_Can_Push:=FALSE;

rolling_have_liao:=FALSE;
Process_3_Can_Push:=FALSE;
Wait_Robot_Push:=FALSE;
Robot2_Push_Finish:=FALSE;
Rolling_Number:=0;
Process_4_Can_Push:=FALSE;
Process_3_Set_Finish:=FALSE;


bak_step:=0;
step:=0;
END_IF
END_PROGRAM

(* Visualisation DEBUG_1
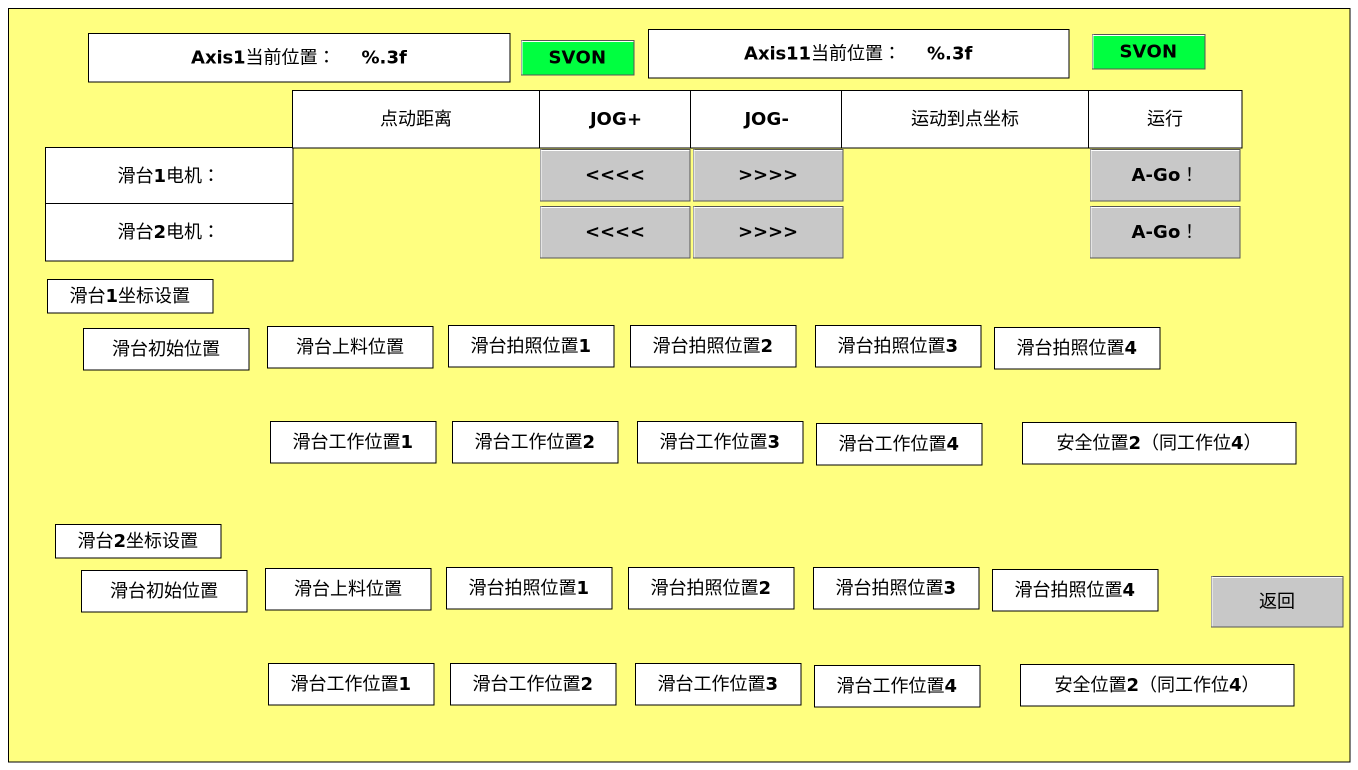
rectangle at (47,145)-(295,203): text "滑台1电机："
rectangle at (47,201)-(295,259): text "滑台2电机："
rectangle at (294,88)-(542,146): text "点动距离"
rectangle at (541,88)-(695,146): text "JOG+"
rectangle at (692,88)-(846,146): text "JOG-"
rectangle at (843,88)-(1091,146): text "运动到点坐标"
rectangle at (1090,88)-(1244,146): text "运行"
button at (542,147)-(692,199): text "<<<<"; taps Axis1_mov_add
button at (542,204)-(692,256): text "<<<<"; taps Axis11_mov_add
button at (695,147)-(845,199): text ">>>>"; taps Axis1_mov_sub
button at (695,204)-(845,256): text ">>>>"; taps Axis11_mov_sub
button at (1092,147)-(1242,199): text "A-Go！"; taps Axis1_mov_line
button at (1092,204)-(1242,256): text "A-Go！"; taps Axis11_mov_line
rectangle at (650,27)-(1071,76): text "Axis11当前位置：    %.3f"; shows D103[10]
rectangle at (90,31)-(512,80): text "Axis1当前位置：    %.3f"; shows D103[0]
rectangle at (49,277)-(215,311): text "滑台1坐标设置"
rectangle at (269,324)-(435,366): text "滑台上料位置"
rectangle at (450,323)-(616,365): text "滑台拍照位置1"
rectangle at (632,323)-(798,365): text "滑台拍照位置2"
rectangle at (817,323)-(983,365): text "滑台拍照位置3"
rectangle at (996,325)-(1162,367): text "滑台拍照位置4"
rectangle at (272,419)-(438,461): text "滑台工作位置1"
rectangle at (454,419)-(620,461): text "滑台工作位置2"
rectangle at (639,419)-(805,461): text "滑台工作位置3"
rectangle at (818,421)-(984,463): text "滑台工作位置4"
rectangle at (1024,420)-(1298,462): text "安全位置2（同工作位4）"
rectangle at (57,522)-(223,556): text "滑台2坐标设置"
rectangle at (85,326)-(251,368): text "滑台初始位置"
rectangle at (267,566)-(433,608): text "滑台上料位置"
rectangle at (448,565)-(614,607): text "滑台拍照位置1"
rectangle at (630,565)-(796,607): text "滑台拍照位置2"
rectangle at (815,565)-(981,607): text "滑台拍照位置3"
rectangle at (994,567)-(1160,609): text "滑台拍照位置4"
rectangle at (270,661)-(436,703): text "滑台工作位置1"
rectangle at (452,661)-(618,703): text "滑台工作位置2"
rectangle at (637,661)-(803,703): text "滑台工作位置3"
rectangle at (816,663)-(982,705): text "滑台工作位置4"
rectangle at (1022,662)-(1296,704): text "安全位置2（同工作位4）"
rectangle at (83,568)-(249,610): text "滑台初始位置"
button at (1213,574)-(1345,625): text "返回"; opens TC_DEBUG
button at (523,38)-(636,73): text "SVON"; toggles Axis1_Poweron
button at (1094,32)-(1207,67): text "SVON"; toggles Axis11_Poweron
1 more shapes without text or variables
25 elements of other kinds (tables, trends, ...) not read
*)

(* Visualisation DEBUG_2
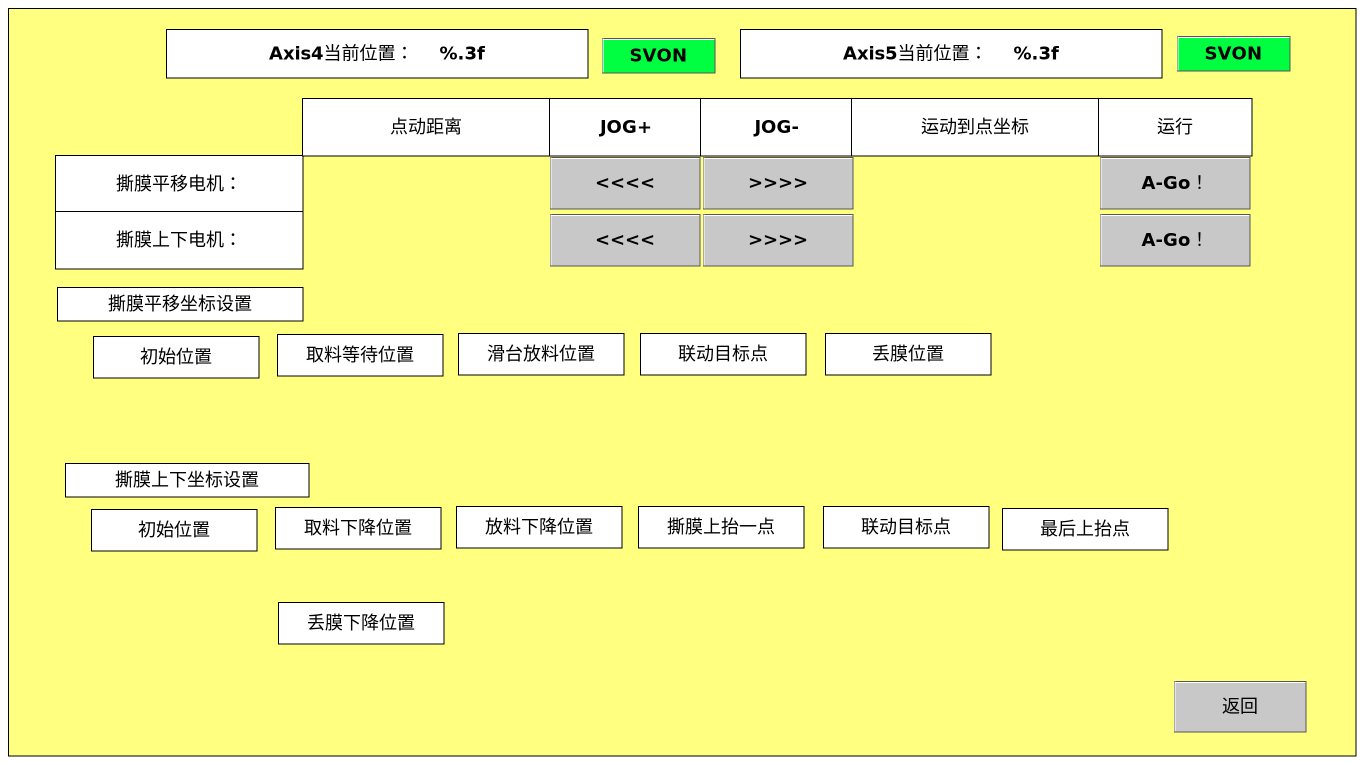
rectangle at (57,155)-(305,213): text "撕膜平移电机："
rectangle at (57,211)-(305,269): text "撕膜上下电机："
rectangle at (304,98)-(552,156): text "点动距离"
rectangle at (551,98)-(705,156): text "JOG+"
rectangle at (702,98)-(856,156): text "JOG-"
rectangle at (853,98)-(1101,156): text "运动到点坐标"
rectangle at (1100,98)-(1254,156): text "运行"
button at (552,157)-(702,209): text "<<<<"; taps Axis4_mov_add
button at (552,214)-(702,266): text "<<<<"; taps Axis5_mov_add
button at (705,157)-(855,209): text ">>>>"; taps Axis4_mov_sub
button at (705,214)-(855,266): text ">>>>"; taps Axis5_mov_sub
button at (1102,157)-(1252,209): text "A-Go！"; taps Axis4_mov_line
button at (1102,214)-(1252,266): text "A-Go！"; taps Axis5_mov_line
rectangle at (59,287)-(305,321): text "撕膜平移坐标设置"
rectangle at (279,334)-(445,376): text "取料等待位置"
rectangle at (460,333)-(626,375): text "滑台放料位置"
rectangle at (642,333)-(808,375): text "联动目标点"
rectangle at (827,333)-(993,375): text "丢膜位置"
rectangle at (67,463)-(311,497): text "撕膜上下坐标设置"
rectangle at (95,336)-(261,378): text "初始位置"
rectangle at (277,507)-(443,549): text "取料下降位置"
rectangle at (458,506)-(624,548): text "放料下降位置"
rectangle at (640,506)-(806,548): text "撕膜上抬一点"
rectangle at (825,506)-(991,548): text "联动目标点"
rectangle at (1004,508)-(1170,550): text "最后上抬点"
rectangle at (280,602)-(446,644): text "丢膜下降位置"
rectangle at (93,509)-(259,551): text "初始位置"
rectangle at (168,29)-(590,78): text "Axis4当前位置：    %.3f"; shows D103[3]
rectangle at (742,29)-(1164,78): text "Axis5当前位置：    %.3f"; shows D103[4]
button at (1176,681)-(1308,732): text "返回"; opens TC_DEBUG
button at (604,38)-(717,73): text "SVON"; toggles Axis4_Poweron
button at (1179,36)-(1292,71): text "SVON"; toggles Axis5_Poweron
1 more shapes without text or variables
15 elements of other kinds (tables, trends, ...) not read
*)

(* Visualisation DEBUG_3
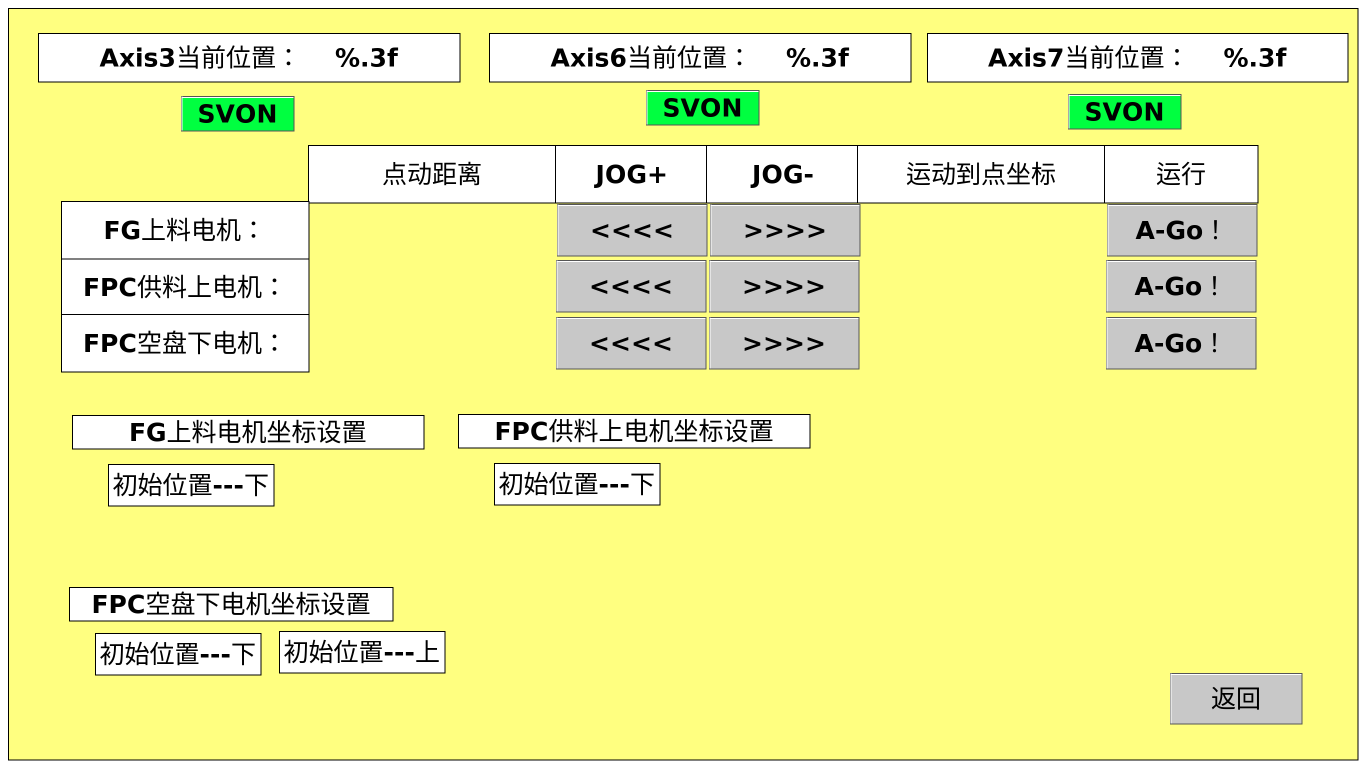
rectangle at (57,256)-(305,314): text "FPC供料上电机："
rectangle at (57,312)-(305,370): text "FPC空盘下电机："
rectangle at (304,143)-(552,201): text "点动距离"
rectangle at (551,143)-(705,201): text "JOG+"
rectangle at (702,143)-(856,201): text "JOG-"
rectangle at (853,143)-(1101,201): text "运动到点坐标"
rectangle at (1100,143)-(1254,201): text "运行"
button at (552,258)-(702,310): text "<<<<"; taps Axis6_mov_add
button at (552,315)-(702,367): text "<<<<"; taps Axis7_mov_add
button at (705,258)-(855,310): text ">>>>"; taps Axis6_mov_sub
button at (705,315)-(855,367): text ">>>>"; taps Axis7_mov_sub
button at (1102,258)-(1252,310): text "A-Go！"; taps Axis6_mov_line
button at (1102,315)-(1252,367): text "A-Go！"; taps Axis7_mov_line
rectangle at (454,412)-(806,446): text "FPC供料上电机坐标设置"
rectangle at (65,585)-(389,619): text "FPC空盘下电机坐标设置"
rectangle at (490,461)-(656,503): text "初始位置---下"
rectangle at (275,629)-(441,671): text "初始位置---上"
rectangle at (91,631)-(257,673): text "初始位置---下"
rectangle at (485,31)-(907,80): text "Axis6当前位置：    %.3f"; shows D103[5]
rectangle at (923,31)-(1344,80): text "Axis7当前位置：    %.3f"; shows D103[6]
rectangle at (57,199)-(305,257): text "FG上料电机："
button at (553,202)-(703,254): text "<<<<"; taps Axis3_mov_add
button at (706,202)-(856,254): text ">>>>"; taps Axis3_mov_sub
button at (1103,202)-(1253,254): text "A-Go！"; taps Axis3_mov_line
rectangle at (68,413)-(420,447): text "FG上料电机坐标设置"
rectangle at (104,462)-(270,504): text "初始位置---下"
button at (1166,671)-(1298,722): text "返回"; opens TC_DEBUG
button at (177,94)-(290,129): text "SVON"; toggles Axis3_Poweron
button at (642,88)-(755,123): text "SVON"; toggles Axis6_Poweron
rectangle at (34,31)-(456,80): text "Axis3当前位置：    %.3f"; shows D103[2]
button at (1064,92)-(1177,127): text "SVON"; toggles Axis7_Poweron
1 more shapes without text or variables
8 elements of other kinds (tables, trends, ...) not read
*)

(* Visualisation DEBUG_4
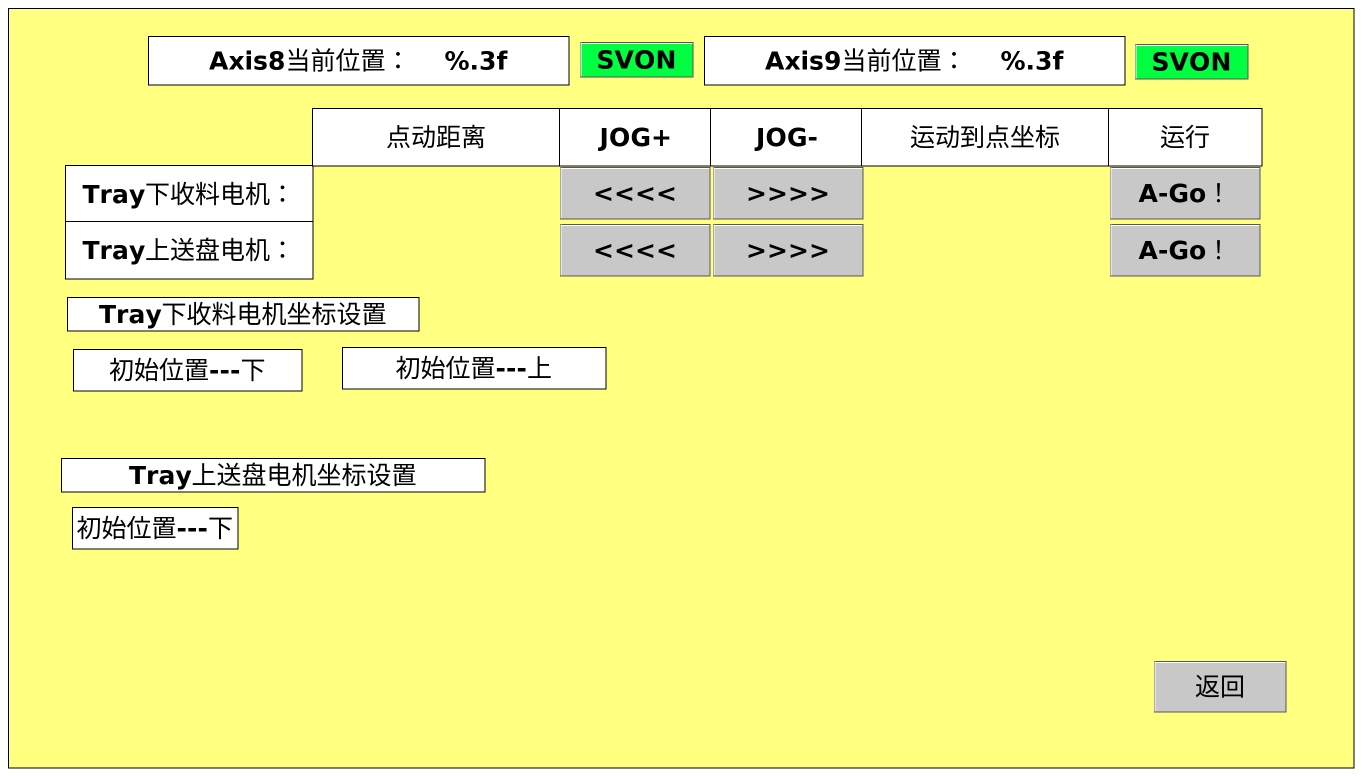
rectangle at (67,165)-(315,223): text "Tray下收料电机："
rectangle at (67,221)-(315,279): text "Tray上送盘电机："
rectangle at (314,108)-(562,166): text "点动距离"
rectangle at (561,108)-(715,166): text "JOG+"
rectangle at (712,108)-(866,166): text "JOG-"
rectangle at (863,108)-(1111,166): text "运动到点坐标"
rectangle at (1110,108)-(1264,166): text "运行"
button at (562,167)-(712,219): text "<<<<"; taps Axis8_mov_add
button at (562,224)-(712,276): text "<<<<"; taps Axis9_mov_add
button at (715,167)-(865,219): text ">>>>"; taps Axis8_mov_sub
button at (715,224)-(865,276): text ">>>>"; taps Axis9_mov_sub
button at (1112,167)-(1262,219): text "A-Go！"; taps Axis8_mov_line
button at (1112,224)-(1262,276): text "A-Go！"; taps Axis9_mov_line
rectangle at (69,297)-(421,331): text "Tray下收料电机坐标设置"
rectangle at (63,458)-(487,492): text "Tray上送盘电机坐标设置"
rectangle at (74,507)-(240,549): text "初始位置---下"
rectangle at (344,347)-(608,389): text "初始位置---上"
rectangle at (75,349)-(304,391): text "初始位置---下"
rectangle at (150,36)-(571,85): text "Axis8当前位置：    %.3f"; shows D103[7]
rectangle at (706,36)-(1127,85): text "Axis9当前位置：    %.3f"; shows D103[8]
button at (1156,661)-(1288,712): text "返回"; opens TC_DEBUG
button at (582,42)-(695,77): text "SVON"; toggles Axis8_Poweron
button at (1137,44)-(1250,79): text "SVON"; toggles Axis9_Poweron
1 more shapes without text or variables
6 elements of other kinds (tables, trends, ...) not read
*)

(* Visualisation DEBUG_5
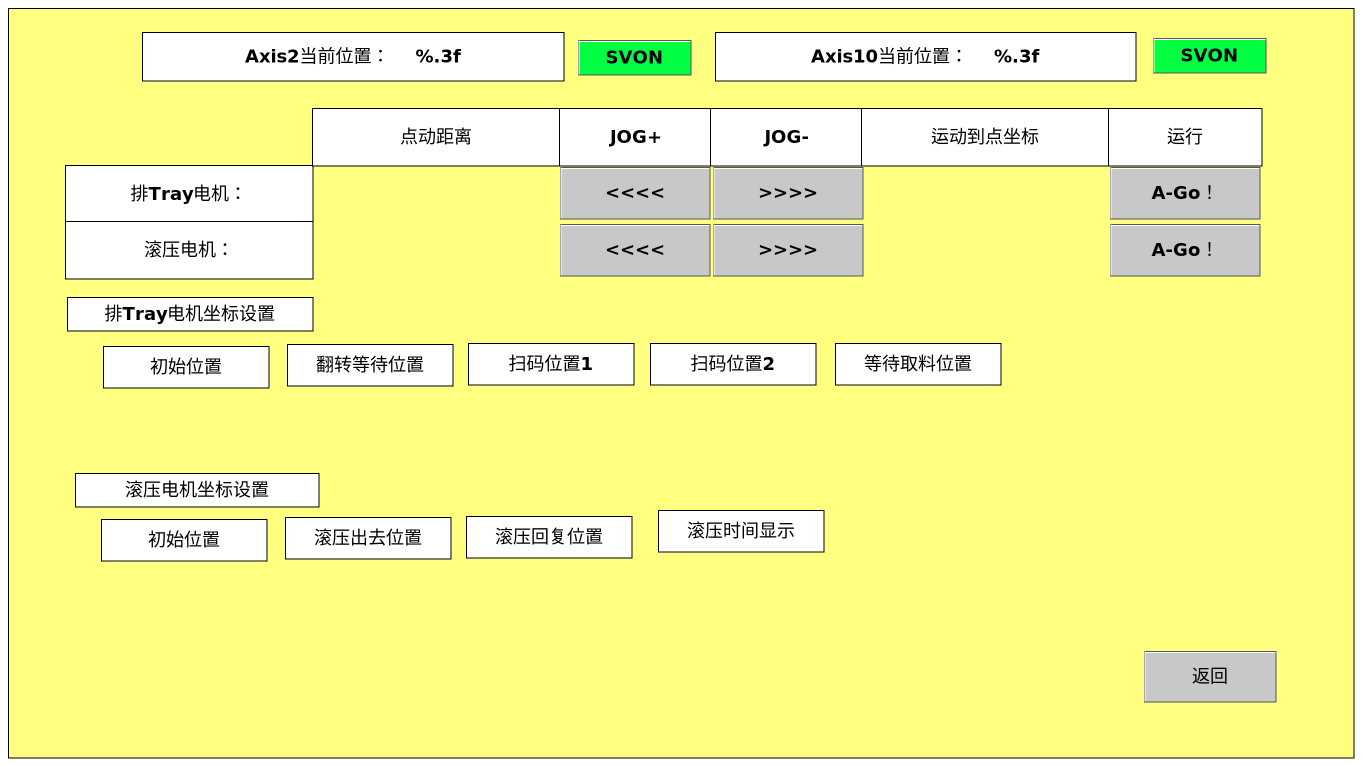
rectangle at (67,165)-(315,223): text "排Tray电机："
rectangle at (67,221)-(315,279): text "滚压电机："
rectangle at (314,108)-(562,166): text "点动距离"
rectangle at (561,108)-(715,166): text "JOG+"
rectangle at (712,108)-(866,166): text "JOG-"
rectangle at (863,108)-(1111,166): text "运动到点坐标"
rectangle at (1110,108)-(1264,166): text "运行"
button at (562,167)-(712,219): text "<<<<"; taps Axis2_mov_add
button at (562,224)-(712,276): text "<<<<"; taps Axis10_mov_add
button at (715,167)-(865,219): text ">>>>"; taps Axis2_mov_sub
button at (715,224)-(865,276): text ">>>>"; taps Axis10_mov_sub
button at (1112,167)-(1262,219): text "A-Go！"; taps Axis2_mov_line
button at (1112,224)-(1262,276): text "A-Go！"; taps Axis10_mov_line
rectangle at (69,297)-(315,331): text "排Tray电机坐标设置"
rectangle at (289,344)-(455,386): text "翻转等待位置"
rectangle at (470,343)-(636,385): text "扫码位置1"
rectangle at (652,343)-(818,385): text "扫码位置2"
rectangle at (837,343)-(1003,385): text "等待取料位置"
rectangle at (77,473)-(321,507): text "滚压电机坐标设置"
rectangle at (105,346)-(271,388): text "初始位置"
rectangle at (287,517)-(453,559): text "滚压出去位置"
rectangle at (468,516)-(634,558): text "滚压回复位置"
rectangle at (103,519)-(269,561): text "初始位置"
rectangle at (717,32)-(1138,81): text "Axis10当前位置：    %.3f"; shows D103[9]
rectangle at (144,32)-(566,81): text "Axis2当前位置：    %.3f"; shows D103[1]
button at (1146,651)-(1278,702): text "返回"; opens TC_DEBUG
button at (580,40)-(693,75): text "SVON"; toggles Axis2_Poweron
button at (1155,38)-(1268,73): text "SVON"; toggles Axis10_Poweron
rectangle at (660,510)-(826,552): text "滚压时间显示"
1 more shapes without text or variables
12 elements of other kinds (tables, trends, ...) not read
*)

(* Visualisation SPECIAL
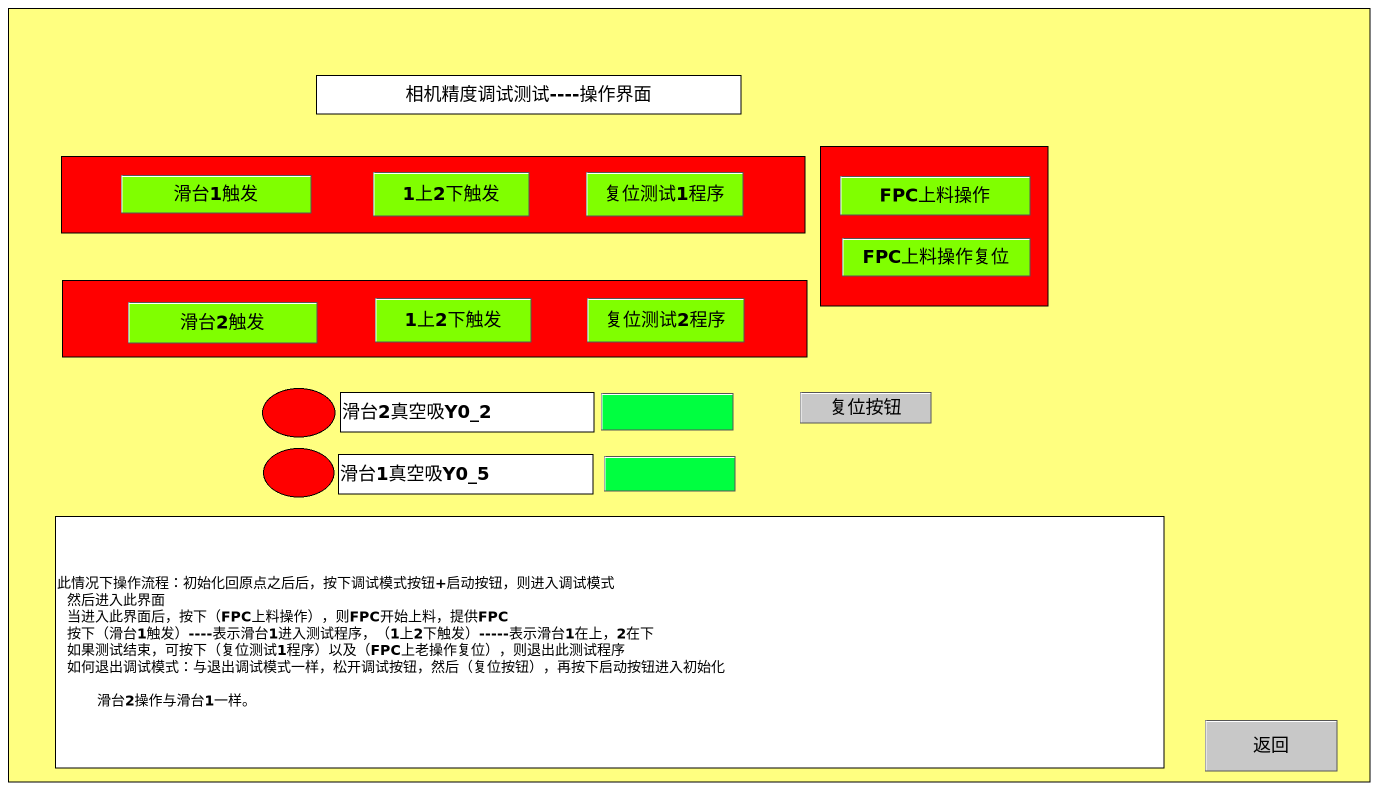
button at (1196,701)-(1328,752): text "返回"; opens TC_DEBUG
rectangle at (46,497)-(1155,749): text "此情况下操作流程：初始化回原点之后后，按下调试模式按钮+启动按钮，则进入调试模式 / 然后进入此界面 / 当进入此界面后，按下（FPC上料操作），则FPC开始上料，提供FPC / 按下（滑台1触发）----表示滑台1进入测试程序，（1上2下触发）-----表示滑台1在上，2在下 / 如果测试结束，可按下（复位测试1程序）以及（FPC上老操作复位），则退出此测试程序 / 如何退出调试模式：与退出调试模式一样，松开调试按钮，然后（复位按钮），再按下启动按钮进入初始化 /  / 滑台2操作与滑台1一样。"
rounded rectangle at (307,56)-(732,95): text "相机精度调试测试----操作界面"
button at (364,153)-(520,197): text "1上2下触发"; taps BU1
button at (577,153)-(734,197): text "复位测试1程序"; taps Rset_Test1
button at (112,156)-(302,194): text "滑台1触发"; toggles Test_Camera_Run_loop
button at (366,279)-(522,323): text "1上2下触发"; taps BU2
button at (578,279)-(735,323): text "复位测试2程序"; taps Rset_Test2
button at (119,283)-(308,324): text "滑台2触发"; toggles Test_Camera_Run_loop1
button at (791,373)-(922,404): text "复位按钮"; taps All_Rset
ellipse at (253,369)-(326,418): alarm colour if Y0_2
rectangle at (331,373)-(585,413): text "滑台2真空吸Y0_2"
ellipse at (254,429)-(325,478): alarm colour if Y0_5
rectangle at (329,435)-(584,475): text "滑台1真空吸Y0_5"
button at (592,374)-(724,411): toggles Y0_2
button at (595,437)-(726,472): toggles Y0_5
button at (831,157)-(1021,196): text "FPC上料操作"; toggles Specila_Feed_FPC
button at (833,219)-(1021,257): text "FPC上料操作复位"; taps Specila_Feed_FPC_OFF
4 more shapes without text or variables
*)

(* Visualisation SPECIAL2
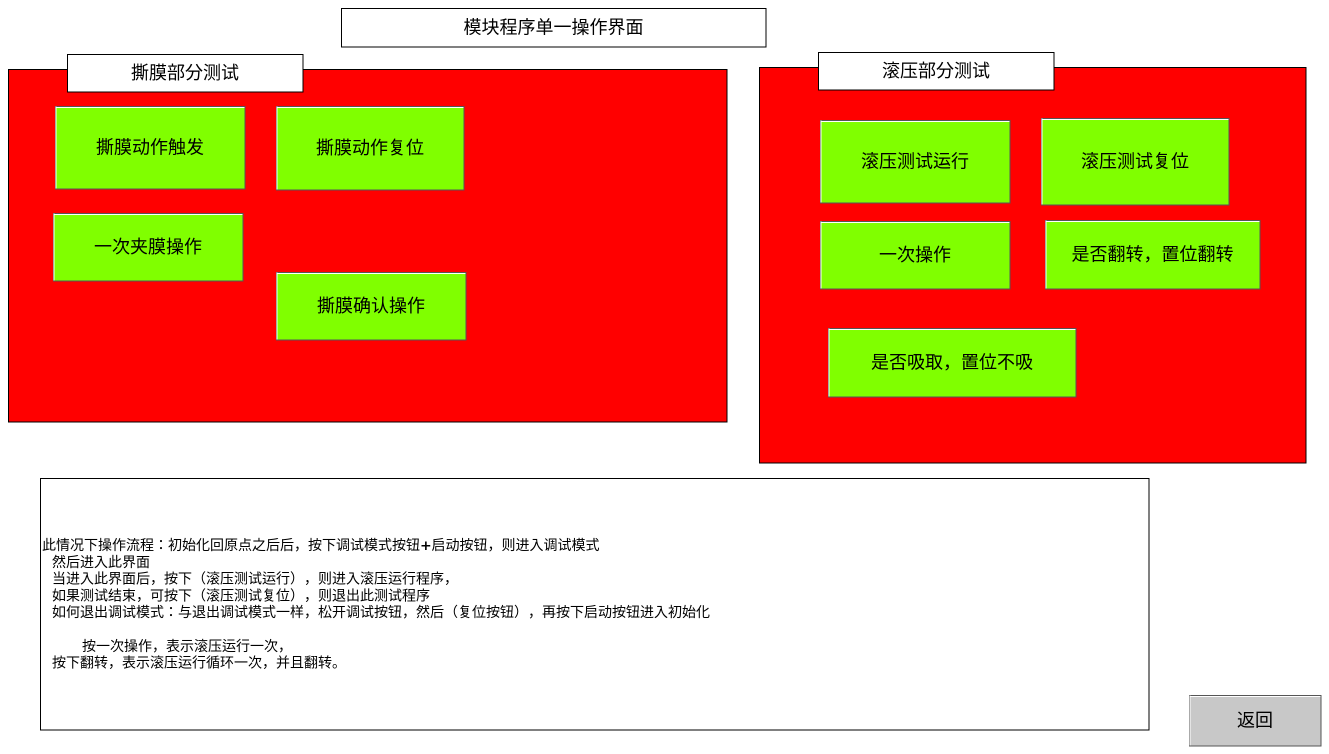
rounded rectangle at (352,13)-(777,52): text "模块程序单一操作界面"
rectangle at (78,59)-(314,97): text "撕膜部分测试"
rectangle at (829,57)-(1065,95): text "滚压部分测试"
button at (1200,700)-(1332,751): text "返回"; opens TC_DEBUG
button at (831,125)-(1021,208): text "滚压测试运行"; toggles Rolling_Part_Run_Test
button at (1052,123)-(1240,210): text "滚压测试复位"; taps Rolling_Part_Run_Test_OFF
button at (1056,225)-(1271,294): text "是否翻转，置位翻转"; toggles Rolling_Pushor_NOT
button at (831,226)-(1021,294): text "一次操作"; toggles Rolling_Once_Run
rectangle at (51,483)-(1160,735): text "此情况下操作流程：初始化回原点之后后，按下调试模式按钮+启动按钮，则进入调试模式 / 然后进入此界面 / 当进入此界面后，按下（滚压测试运行），则进入滚压运行程序， / 如果测试结束，可按下（滚压测试复位），则退出此测试程序 / 如何退出调试模式：与退出调试模式一样，松开调试按钮，然后（复位按钮），再按下启动按钮进入初始化 /  / 按一次操作，表示滚压运行一次， / 按下翻转，表示滚压运行循环一次，并且翻转。"
button at (839,333)-(1087,402): text "是否吸取，置位不吸"; toggles Empty_Pro
button at (66,111)-(256,194): text "撕膜动作触发"; toggles Film_Test
button at (287,111)-(475,195): text "撕膜动作复位"; taps Film_Test_OFF
button at (64,218)-(254,286): text "一次夹膜操作"; taps Film_Once_Run
button at (287,277)-(477,345): text "撕膜确认操作"; taps Qurensimo
2 more shapes without text or variables
*)

(* Visualisation TC_C
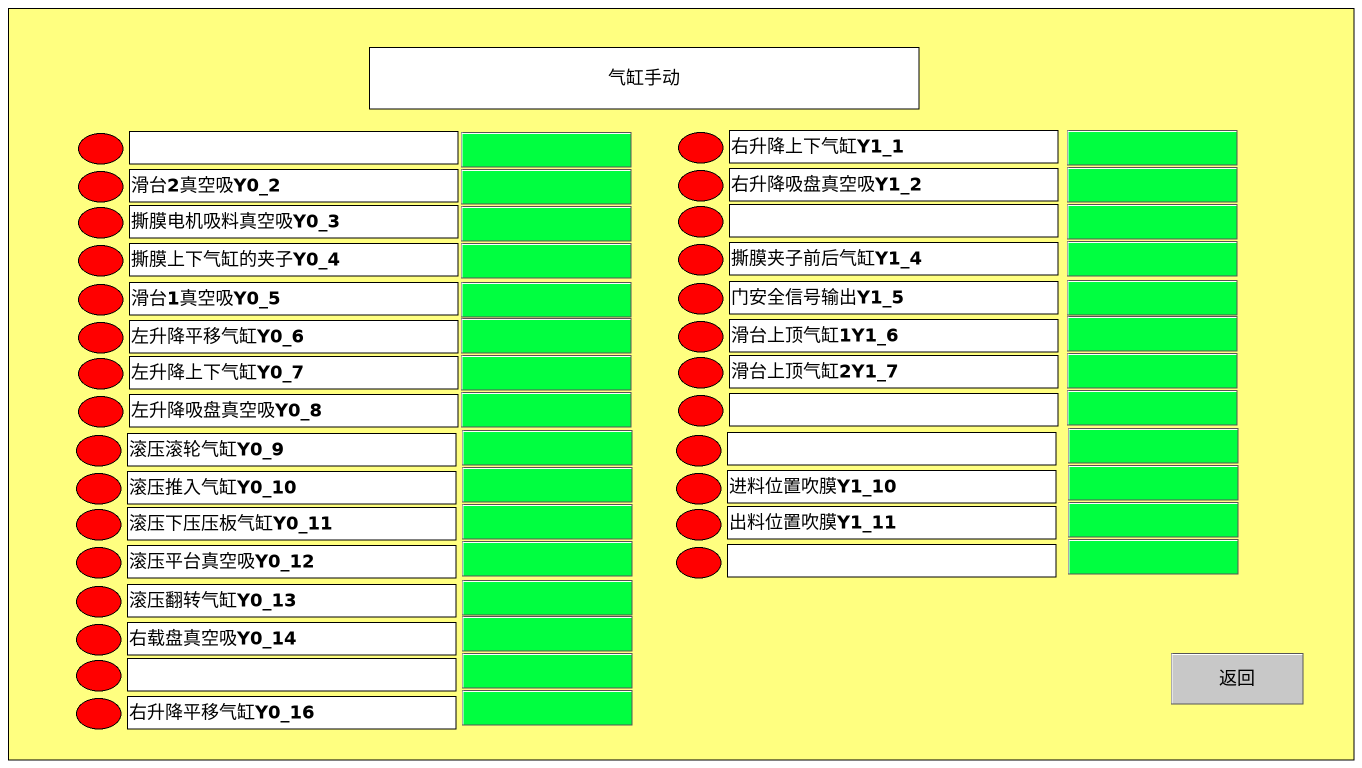
button at (1171,653)-(1303,704): text "返回"; opens TC_DEBUG
rounded rectangle at (369,47)-(919,109): text "气缸手动"
ellipse at (78,133)-(123,164): alarm colour if Y0_1
ellipse at (78,171)-(123,202): alarm colour if Y0_2
rectangle at (129,169)-(458,202): text "滑台2真空吸Y0_2"
ellipse at (78,207)-(123,238): alarm colour if Y0_3
rectangle at (129,205)-(458,238): text "撕膜电机吸料真空吸Y0_3"
ellipse at (78,245)-(123,276): alarm colour if Y0_4
rectangle at (129,243)-(458,276): text "撕膜上下气缸的夹子Y0_4"
ellipse at (78,284)-(123,315): alarm colour if Y0_5
rectangle at (129,282)-(458,315): text "滑台1真空吸Y0_5"
ellipse at (78,322)-(123,353): alarm colour if Y0_6
rectangle at (129,320)-(458,353): text "左升降平移气缸Y0_6"
ellipse at (78,358)-(123,389): alarm colour if Y0_7
rectangle at (129,356)-(458,389): text "左升降上下气缸Y0_7"
ellipse at (78,396)-(123,427): alarm colour if Y0_8
rectangle at (129,394)-(458,427): text "左升降吸盘真空吸Y0_8"
ellipse at (76,435)-(121,466): alarm colour if Y0_9
rectangle at (127,433)-(456,466): text "滚压滚轮气缸Y0_9"
ellipse at (76,473)-(121,504): alarm colour if Y0_10
rectangle at (127,471)-(456,504): text "滚压推入气缸Y0_10"
ellipse at (76,509)-(121,540): alarm colour if Y0_11
rectangle at (127,507)-(456,540): text "滚压下压压板气缸Y0_11"
ellipse at (76,547)-(121,578): alarm colour if Y0_12
rectangle at (127,545)-(456,578): text "滚压平台真空吸Y0_12"
ellipse at (76,586)-(121,617): alarm colour if Y0_13
rectangle at (127,584)-(456,617): text "滚压翻转气缸Y0_13"
ellipse at (76,624)-(121,655): alarm colour if Y0_14
rectangle at (127,622)-(456,655): text "右载盘真空吸Y0_14"
ellipse at (76,660)-(121,691): alarm colour if Y0_15
ellipse at (76,698)-(121,729): alarm colour if Y0_16
rectangle at (127,696)-(456,729): text "右升降平移气缸Y0_16"
ellipse at (678,132)-(723,163): alarm colour if Y1_1
rectangle at (729,130)-(1058,163): text "右升降上下气缸Y1_1"
ellipse at (678,170)-(723,201): alarm colour if Y1_2
rectangle at (729,168)-(1058,201): text "右升降吸盘真空吸Y1_2"
ellipse at (678,206)-(723,237): alarm colour if Y1_3
ellipse at (678,244)-(723,275): alarm colour if Y1_4
rectangle at (729,242)-(1058,275): text "撕膜夹子前后气缸Y1_4"
ellipse at (678,283)-(723,314): alarm colour if Y1_5
rectangle at (729,281)-(1058,314): text "门安全信号输出Y1_5"
ellipse at (678,321)-(723,352): alarm colour if Y1_6
rectangle at (729,319)-(1058,352): text "滑台上顶气缸1Y1_6"
ellipse at (678,357)-(723,388): alarm colour if Y1_7
rectangle at (729,355)-(1058,388): text "滑台上顶气缸2Y1_7"
ellipse at (678,395)-(723,426): alarm colour if Y1_8
ellipse at (676,435)-(721,466): alarm colour if Y1_9
ellipse at (676,473)-(721,504): alarm colour if Y1_10
rectangle at (727,470)-(1056,503): text "进料位置吹膜Y1_10"
ellipse at (676,509)-(721,540): alarm colour if Y1_11
rectangle at (727,506)-(1056,539): text "出料位置吹膜Y1_11"
ellipse at (676,547)-(721,578): alarm colour if Y1_12
button at (461,132)-(631,167): toggles Y0_1
button at (461,169)-(631,204): toggles Y0_2
button at (461,206)-(631,241): toggles Y0_3
button at (461,243)-(631,278): toggles Y0_4
button at (461,282)-(631,317): toggles Y0_5
button at (461,318)-(631,353): toggles Y0_6
button at (461,355)-(631,390): toggles Y0_7
button at (461,392)-(631,427): toggles Y0_8
button at (462,430)-(632,465): toggles Y0_9
button at (462,467)-(632,502): toggles Y0_10
button at (462,504)-(632,539): toggles Y0_11
button at (462,541)-(632,576): toggles Y0_12
button at (462,580)-(632,615): toggles Y0_13
button at (462,616)-(632,651): toggles Y0_14
button at (462,653)-(632,688): toggles Y0_15
button at (462,690)-(632,725): toggles Y0_16
button at (1067,130)-(1237,165): toggles Y1_1
button at (1067,167)-(1237,202): toggles Y1_2
button at (1067,204)-(1237,239): toggles Y1_3
button at (1067,241)-(1237,276): toggles Y1_4
button at (1067,280)-(1237,315): toggles Y1_5
button at (1067,316)-(1237,351): toggles Y1_6
button at (1067,353)-(1237,388): toggles Y1_7
button at (1067,390)-(1237,425): toggles Y1_8
button at (1068,428)-(1238,463): toggles Y1_9
button at (1068,465)-(1238,500): toggles Y1_10
button at (1068,502)-(1238,537): toggles Y1_11
button at (1068,539)-(1238,574): toggles Y1_12
7 more shapes without text or variables
*)

(* Visualisation TC_DEBUG
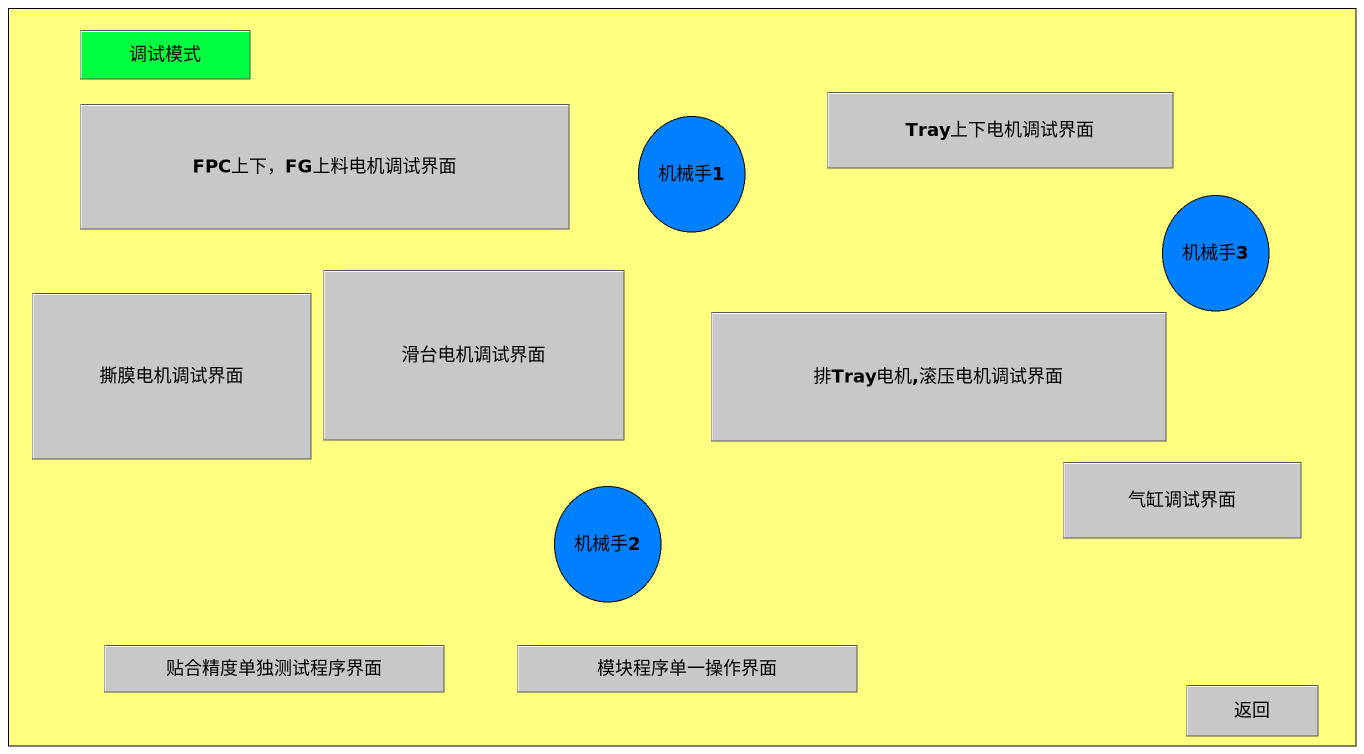
button at (323,276)-(624,446): text "滑台电机调试界面"; opens DEBUG_1
button at (32,299)-(311,465): text "撕膜电机调试界面"; opens DEBUG_2
button at (80,110)-(569,235): text "FPC上下，FG上料电机调试界面"; opens DEBUG_3
button at (827,98)-(1173,174): text "Tray上下电机调试界面"; opens DEBUG_4
button at (711,318)-(1166,447): text "排Tray电机,滚压电机调试界面"; opens DEBUG_5
button at (1063,468)-(1301,544): text "气缸调试界面"; opens TC_C
ellipse at (638,122)-(745,238): text "机械手1"
ellipse at (554,492)-(661,608): text "机械手2"
ellipse at (1162,201)-(1269,317): text "机械手3"
button at (1186,691)-(1318,742): text "返回"; opens TC_VIEW
button at (80,36)-(250,85): text "调试模式"; toggles Debug_Model
button at (104,651)-(444,698): text "贴合精度单独测试程序界面"; opens SPECIAL
button at (517,651)-(857,698): text "模块程序单一操作界面"; opens SPECIAL2
1 more shapes without text or variables
*)

(* Visualisation TC_HMI
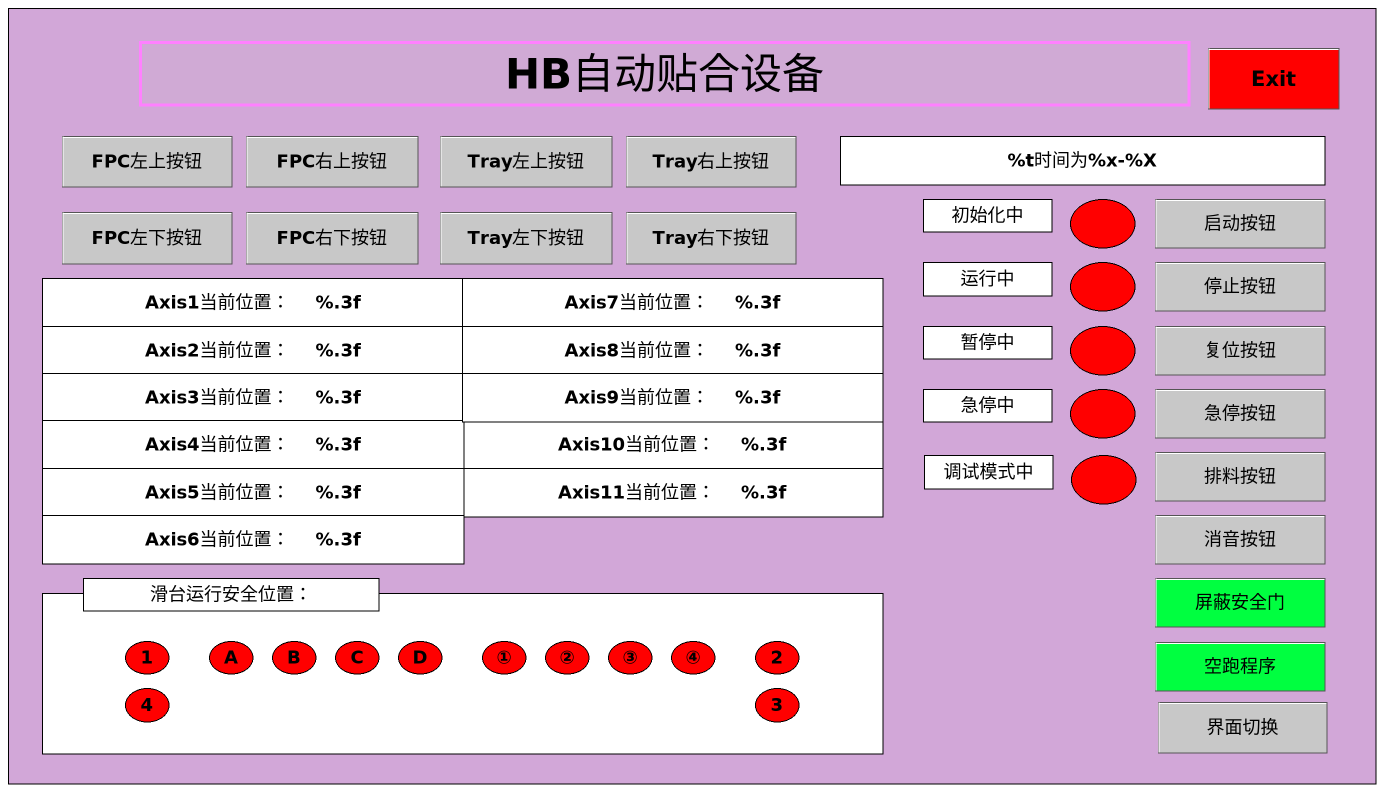
rectangle at (832,118)-(1317,167): text "%t时间为%x-%X"
button at (1147,181)-(1317,230): text "启动按钮"; taps All_Start
button at (1147,244)-(1317,293): text "停止按钮"; taps All_Stop
button at (1147,308)-(1317,357): text "复位按钮"; taps All_Rset
button at (1147,371)-(1317,420): text "急停按钮"; toggles Total_Emergency
button at (1147,434)-(1317,483): text "排料按钮"; toggles Discharge_Button
rectangle at (915,181)-(1044,214): text "初始化中"
rectangle at (915,244)-(1044,278): text "运行中"
rectangle at (915,308)-(1044,341): text "暂停中"
ellipse at (1062,371)-(1127,420): alarm colour if Total_Emergency
rectangle at (915,371)-(1044,404): text "急停中"
ellipse at (1062,244)-(1127,293): alarm colour if runing
ellipse at (1062,308)-(1127,357): alarm colour if Total_Pause
button at (1147,497)-(1317,546): text "消音按钮"; taps Silencer_Button
button at (1147,560)-(1317,609): text "屏蔽安全门"; toggles Shield_Door
button at (1147,624)-(1317,673): text "空跑程序"; toggles Empty_Pro
rectangle at (454,402)-(875,451): text "Axis10当前位置：    %.3f"; shows D103[9]
rectangle at (454,450)-(875,499): text "Axis11当前位置：    %.3f"; shows D103[10]
rectangle at (34,260)-(456,309): text "Axis1当前位置：    %.3f"; shows D103[0]
rectangle at (34,308)-(456,357): text "Axis2当前位置：    %.3f"; shows D103[1]
rectangle at (34,355)-(456,404): text "Axis3当前位置：    %.3f"; shows D103[2]
rectangle at (34,402)-(456,451): text "Axis4当前位置：    %.3f"; shows D103[3]
rectangle at (34,450)-(456,499): text "Axis5当前位置：    %.3f"; shows D103[4]
rectangle at (34,497)-(456,546): text "Axis6当前位置：    %.3f"; shows D103[5]
rectangle at (454,260)-(875,309): text "Axis7当前位置：    %.3f"; shows D103[6]
rectangle at (454,308)-(875,357): text "Axis8当前位置：    %.3f"; shows D103[7]
rectangle at (454,355)-(875,404): text "Axis9当前位置：    %.3f"; shows D103[8]
button at (54,118)-(224,169): text "FPC左上按钮"; taps Left_Down_Button
button at (238,194)-(410,246): text "FPC右下按钮"; taps Feed_Left_Button1
button at (238,118)-(410,169): text "FPC右上按钮"; taps Left_UP_Button
button at (54,194)-(224,246): text "FPC左下按钮"; taps Feed_Left_Button2
button at (432,118)-(604,169): text "Tray左上按钮"; taps Right_Up_Button
button at (618,194)-(788,246): text "Tray右下按钮"; taps Feed_Right_Button1
button at (618,118)-(788,169): text "Tray右上按钮"; taps Right_Down_Button
button at (432,194)-(604,246): text "Tray左下按钮"; taps Feed_Right_Button2
ellipse at (1062,181)-(1127,230): alarm colour if IsIniing
rectangle at (131,23)-(1182,88): text "HB自动贴合设备"
ellipse at (117,623)-(161,656): text "1"; alarm colour if Positive1_Safe
ellipse at (747,670)-(791,704): text "3"; alarm colour if Positive3_Safe
ellipse at (117,670)-(161,704): text "4"; alarm colour if Positive4_Safe
ellipse at (747,623)-(791,656): text "2"; alarm colour if Positive2_Safe
ellipse at (390,623)-(434,656): text "D"; alarm colour if Positive_Camera_Safe4
ellipse at (201,623)-(245,656): text "A"; alarm colour if Positive_Camera_Safe1
ellipse at (264,623)-(308,656): text "B"; alarm colour if Positive_Camera_Safe2
ellipse at (327,623)-(371,656): text "C"; alarm colour if Positive_Camera_Safe3
ellipse at (663,623)-(707,656): text "④"; alarm colour if Positive_Fit_Safe4
ellipse at (474,623)-(518,656): text "①"; alarm colour if Positive_Fit_Safe1
ellipse at (537,623)-(581,656): text "②"; alarm colour if Positive_Fit_Safe2
ellipse at (600,623)-(644,656): text "③"; alarm colour if Positive_Fit_Safe3
rectangle at (75,560)-(371,593): text "滑台运行安全位置："
button at (1200,30)-(1331,91): text "Exit"; runs INTERN EXITPROGRAM
button at (1150,684)-(1319,735): text "界面切换"; opens TC_VIEW
rectangle at (916,437)-(1045,471): text "调试模式中"
ellipse at (1063,437)-(1128,486): alarm colour if Debug_Model
2 more shapes without text or variables
*)

(* Visualisation TC_IO1
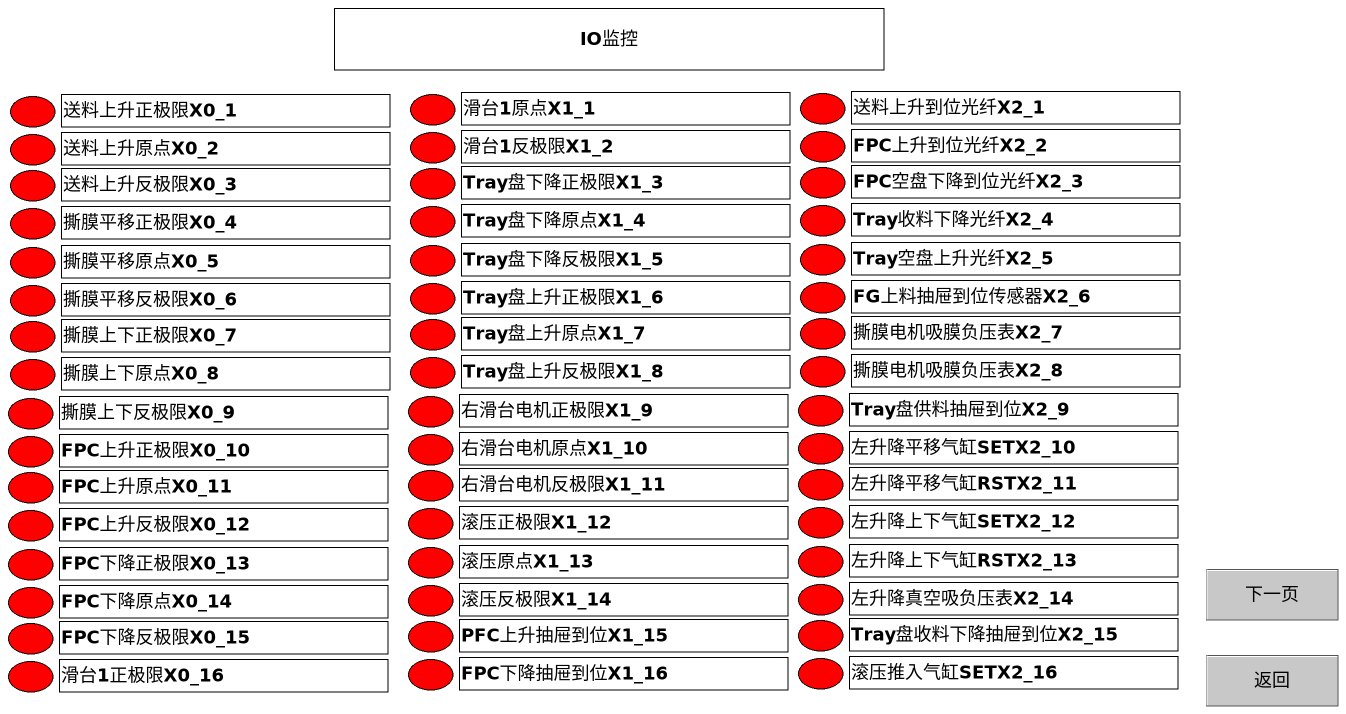
button at (1221,675)-(1353,726): text "返回"; opens TC_VIEW
rounded rectangle at (349,28)-(899,90): text "IO监控"
ellipse at (25,116)-(70,147): alarm colour if X0_1
rectangle at (76,114)-(405,147): text "送料上升正极限X0_1"
ellipse at (25,154)-(70,185): alarm colour if X0_2
rectangle at (76,152)-(405,185): text "送料上升原点X0_2"
ellipse at (25,190)-(70,221): alarm colour if X0_3
rectangle at (76,188)-(405,221): text "送料上升反极限X0_3"
ellipse at (25,228)-(70,259): alarm colour if X0_4
rectangle at (76,226)-(405,259): text "撕膜平移正极限X0_4"
ellipse at (25,267)-(70,298): alarm colour if X0_5
rectangle at (76,265)-(405,298): text "撕膜平移原点X0_5"
ellipse at (25,305)-(70,336): alarm colour if X0_6
rectangle at (76,303)-(405,336): text "撕膜平移反极限X0_6"
ellipse at (25,341)-(70,372): alarm colour if X0_7
rectangle at (76,339)-(405,372): text "撕膜上下正极限X0_7"
ellipse at (25,379)-(70,410): alarm colour if X0_8
rectangle at (76,377)-(405,410): text "撕膜上下原点X0_8"
ellipse at (23,418)-(68,449): alarm colour if X0_9
rectangle at (74,416)-(403,449): text "撕膜上下反极限X0_9"
ellipse at (23,456)-(68,487): alarm colour if X0_10
rectangle at (74,454)-(403,487): text "FPC上升正极限X0_10"
ellipse at (23,492)-(68,523): alarm colour if X0_11
rectangle at (74,490)-(403,523): text "FPC上升原点X0_11"
ellipse at (23,530)-(68,561): alarm colour if X0_12
rectangle at (74,528)-(403,561): text "FPC上升反极限X0_12"
ellipse at (23,569)-(68,600): alarm colour if X0_13
rectangle at (74,567)-(403,600): text "FPC下降正极限X0_13"
ellipse at (23,607)-(68,638): alarm colour if X0_14
rectangle at (74,605)-(403,638): text "FPC下降原点X0_14"
ellipse at (23,643)-(68,674): alarm colour if X0_15
rectangle at (74,641)-(403,674): text "FPC下降反极限X0_15"
ellipse at (23,681)-(68,712): alarm colour if X0_16
rectangle at (74,679)-(403,712): text "滑台1正极限X0_16"
button at (1221,589)-(1353,640): text "下一页"; opens TC_IO2
ellipse at (425,114)-(470,145): alarm colour if X1_1
rectangle at (476,112)-(805,145): text "滑台1原点X1_1"
ellipse at (425,152)-(470,183): alarm colour if X1_2
rectangle at (476,150)-(805,183): text "滑台1反极限X1_2"
ellipse at (425,188)-(470,219): alarm colour if X1_3
rectangle at (476,186)-(805,219): text "Tray盘下降正极限X1_3"
ellipse at (425,226)-(470,257): alarm colour if X1_4
rectangle at (476,224)-(805,257): text "Tray盘下降原点X1_4"
ellipse at (425,265)-(470,296): alarm colour if X1_5
rectangle at (476,263)-(805,296): text "Tray盘下降反极限X1_5"
ellipse at (425,303)-(470,334): alarm colour if X1_6
rectangle at (476,301)-(805,334): text "Tray盘上升正极限X1_6"
ellipse at (425,339)-(470,370): alarm colour if X1_7
rectangle at (476,337)-(805,370): text "Tray盘上升原点X1_7"
ellipse at (425,377)-(470,408): alarm colour if X1_8
rectangle at (476,375)-(805,408): text "Tray盘上升反极限X1_8"
ellipse at (423,416)-(468,447): alarm colour if X1_9
rectangle at (474,414)-(803,447): text "右滑台电机正极限X1_9"
ellipse at (423,454)-(468,485): alarm colour if X1_10
rectangle at (474,452)-(803,485): text "右滑台电机原点X1_10"
ellipse at (423,490)-(468,521): alarm colour if X1_11
rectangle at (474,488)-(803,521): text "右滑台电机反极限X1_11"
ellipse at (423,528)-(468,559): alarm colour if X1_12
rectangle at (474,526)-(803,559): text "滚压正极限X1_12"
ellipse at (423,567)-(468,598): alarm colour if X1_13
rectangle at (474,565)-(803,598): text "滚压原点X1_13"
ellipse at (423,605)-(468,636): alarm colour if X1_14
rectangle at (474,603)-(803,636): text "滚压反极限X1_14"
ellipse at (423,641)-(468,672): alarm colour if X1_15
rectangle at (474,639)-(803,672): text "PFC上升抽屉到位X1_15"
ellipse at (423,679)-(468,710): alarm colour if X1_16
rectangle at (474,677)-(803,710): text "FPC下降抽屉到位X1_16"
ellipse at (815,113)-(860,144): alarm colour if X2_1
rectangle at (866,111)-(1195,144): text "送料上升到位光纤X2_1"
ellipse at (815,151)-(860,182): alarm colour if X2_2
rectangle at (866,149)-(1195,182): text "FPC上升到位光纤X2_2"
ellipse at (815,187)-(860,218): alarm colour if X2_3
rectangle at (866,185)-(1195,218): text "FPC空盘下降到位光纤X2_3"
ellipse at (815,225)-(860,256): alarm colour if X2_4
rectangle at (866,223)-(1195,256): text "Tray收料下降光纤X2_4"
ellipse at (815,264)-(860,295): alarm colour if X2_5
rectangle at (866,262)-(1195,295): text "Tray空盘上升光纤X2_5"
ellipse at (815,302)-(860,333): alarm colour if X2_6
rectangle at (866,300)-(1195,333): text "FG上料抽屉到位传感器X2_6"
ellipse at (815,338)-(860,369): alarm colour if X2_7
rectangle at (866,336)-(1195,369): text "撕膜电机吸膜负压表X2_7"
ellipse at (815,376)-(860,407): alarm colour if X2_8
rectangle at (866,374)-(1195,407): text "撕膜电机吸膜负压表X2_8"
ellipse at (813,415)-(858,446): alarm colour if X2_9
rectangle at (864,413)-(1193,446): text "Tray盘供料抽屉到位X2_9"
ellipse at (813,453)-(858,484): alarm colour if X2_10
rectangle at (864,451)-(1193,484): text "左升降平移气缸SETX2_10"
ellipse at (813,489)-(858,520): alarm colour if X2_11
rectangle at (864,487)-(1193,520): text "左升降平移气缸RSTX2_11"
ellipse at (813,527)-(858,558): alarm colour if X2_12
rectangle at (864,525)-(1193,558): text "左升降上下气缸SETX2_12"
ellipse at (813,566)-(858,597): alarm colour if X2_13
rectangle at (864,564)-(1193,597): text "左升降上下气缸RSTX2_13"
ellipse at (813,604)-(858,635): alarm colour if X2_14
rectangle at (864,602)-(1193,635): text "左升降真空吸负压表X2_14"
ellipse at (813,640)-(858,671): alarm colour if X2_15
rectangle at (864,638)-(1193,671): text "Tray盘收料下降抽屉到位X2_15"
ellipse at (813,678)-(858,709): alarm colour if X2_16
rectangle at (864,676)-(1193,709): text "滚压推入气缸SETX2_16"
*)

(* Visualisation TC_IO2
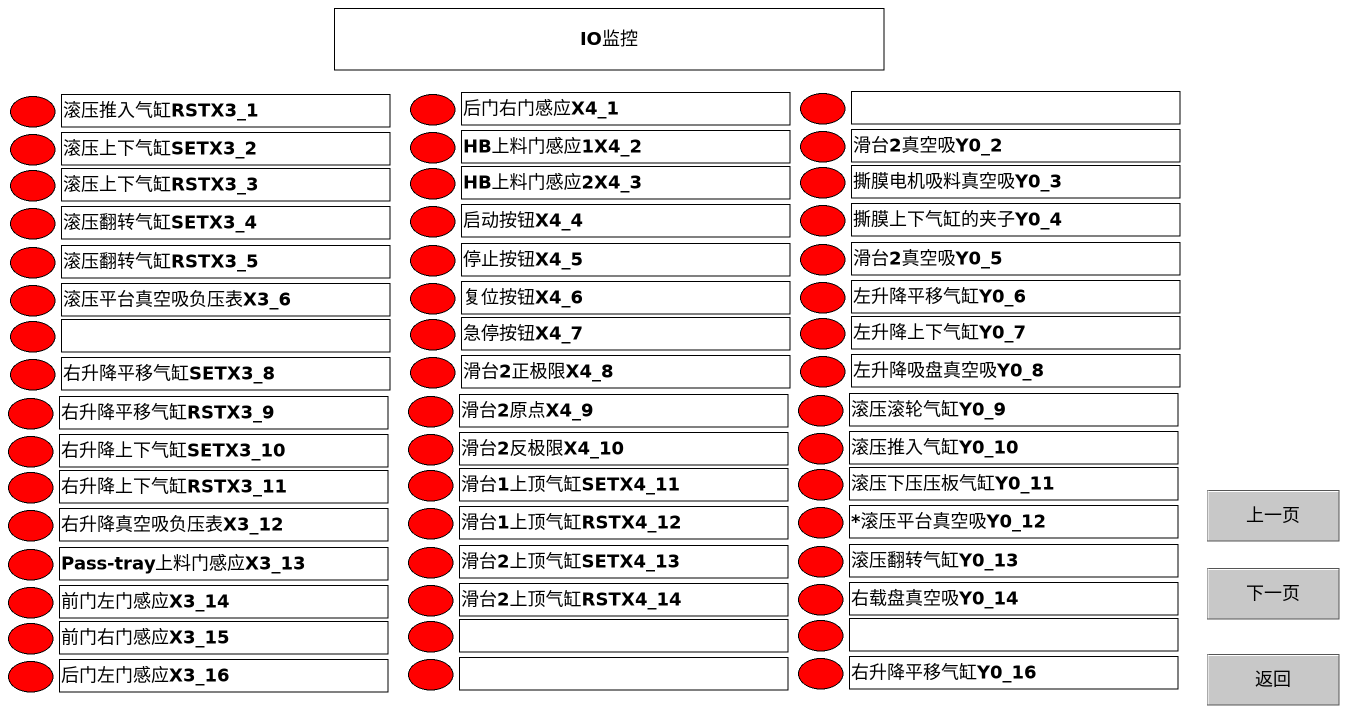
button at (1221,685)-(1353,736): text "返回"; opens TC_VIEW
button at (1221,599)-(1353,650): text "下一页"; opens TC_IO3
button at (1221,521)-(1353,572): text "上一页"; opens TC_IO1
rounded rectangle at (348,39)-(898,101): text "IO监控"
ellipse at (24,127)-(69,158): alarm colour if X3_1
rectangle at (75,125)-(404,158): text "滚压推入气缸RSTX3_1"
ellipse at (24,165)-(69,196): alarm colour if X3_2
rectangle at (75,163)-(404,196): text "滚压上下气缸SETX3_2"
ellipse at (24,201)-(69,232): alarm colour if X3_3
rectangle at (75,199)-(404,232): text "滚压上下气缸RSTX3_3"
ellipse at (24,239)-(69,270): alarm colour if X3_4
rectangle at (75,237)-(404,270): text "滚压翻转气缸SETX3_4"
ellipse at (24,278)-(69,309): alarm colour if X3_5
rectangle at (75,276)-(404,309): text "滚压翻转气缸RSTX3_5"
ellipse at (24,316)-(69,347): alarm colour if X3_6
rectangle at (75,314)-(404,347): text "滚压平台真空吸负压表X3_6"
ellipse at (24,352)-(69,383): alarm colour if X3_7
ellipse at (24,390)-(69,421): alarm colour if X3_8
rectangle at (75,388)-(404,421): text "右升降平移气缸SETX3_8"
ellipse at (22,429)-(67,460): alarm colour if X3_9
rectangle at (73,427)-(402,460): text "右升降平移气缸RSTX3_9"
ellipse at (22,467)-(67,498): alarm colour if X3_10
rectangle at (73,465)-(402,498): text "右升降上下气缸SETX3_10"
ellipse at (22,503)-(67,534): alarm colour if X3_11
rectangle at (73,501)-(402,534): text "右升降上下气缸RSTX3_11"
ellipse at (22,541)-(67,572): alarm colour if X3_12
rectangle at (73,539)-(402,572): text "右升降真空吸负压表X3_12"
ellipse at (22,580)-(67,611): alarm colour if X3_13
rectangle at (73,578)-(402,611): text "Pass-tray上料门感应X3_13"
ellipse at (22,618)-(67,649): alarm colour if X3_14
rectangle at (73,616)-(402,649): text "前门左门感应X3_14"
ellipse at (22,654)-(67,685): alarm colour if X3_15
rectangle at (73,652)-(402,685): text "前门右门感应X3_15"
ellipse at (22,692)-(67,723): alarm colour if X3_16
rectangle at (73,690)-(402,723): text "后门左门感应X3_16"
ellipse at (424,125)-(469,156): alarm colour if X4_1
rectangle at (475,123)-(804,156): text "后门右门感应X4_1"
ellipse at (424,163)-(469,194): alarm colour if X4_2
rectangle at (475,161)-(804,194): text "HB上料门感应1X4_2"
ellipse at (424,199)-(469,230): alarm colour if X4_3
rectangle at (475,197)-(804,230): text "HB上料门感应2X4_3"
ellipse at (424,237)-(469,268): alarm colour if X4_4
rectangle at (475,235)-(804,268): text "启动按钮X4_4"
ellipse at (424,276)-(469,307): alarm colour if X4_5
rectangle at (475,274)-(804,307): text "停止按钮X4_5"
ellipse at (424,314)-(469,345): alarm colour if X4_6
rectangle at (475,312)-(804,345): text "复位按钮X4_6"
ellipse at (424,350)-(469,381): alarm colour if X4_7
rectangle at (475,348)-(804,381): text "急停按钮X4_7"
ellipse at (424,388)-(469,419): alarm colour if X4_8
rectangle at (475,386)-(804,419): text "滑台2正极限X4_8"
ellipse at (422,427)-(467,458): alarm colour if X4_9
rectangle at (473,425)-(802,458): text "滑台2原点X4_9"
ellipse at (422,465)-(467,496): alarm colour if X4_10
rectangle at (473,463)-(802,496): text "滑台2反极限X4_10"
ellipse at (422,501)-(467,532): alarm colour if X4_11
rectangle at (473,499)-(802,532): text "滑台1上顶气缸SETX4_11"
ellipse at (422,539)-(467,570): alarm colour if X4_12
rectangle at (473,537)-(802,570): text "滑台1上顶气缸RSTX4_12"
ellipse at (422,578)-(467,609): alarm colour if X4_13
rectangle at (473,576)-(802,609): text "滑台2上顶气缸SETX4_13"
ellipse at (422,616)-(467,647): alarm colour if X4_14
rectangle at (473,614)-(802,647): text "滑台2上顶气缸RSTX4_14"
ellipse at (422,652)-(467,683): alarm colour if X4_15
ellipse at (422,690)-(467,721): alarm colour if X4_16
ellipse at (814,124)-(859,155): alarm colour if Y0_1
ellipse at (814,162)-(859,193): alarm colour if Y0_2
rectangle at (865,160)-(1194,193): text "滑台2真空吸Y0_2"
ellipse at (814,198)-(859,229): alarm colour if Y0_3
rectangle at (865,196)-(1194,229): text "撕膜电机吸料真空吸Y0_3"
ellipse at (814,236)-(859,267): alarm colour if Y0_4
rectangle at (865,234)-(1194,267): text "撕膜上下气缸的夹子Y0_4"
ellipse at (814,275)-(859,306): alarm colour if Y0_5
rectangle at (865,273)-(1194,306): text "滑台2真空吸Y0_5"
ellipse at (814,313)-(859,344): alarm colour if Y0_6
rectangle at (865,311)-(1194,344): text "左升降平移气缸Y0_6"
ellipse at (814,349)-(859,380): alarm colour if Y0_7
rectangle at (865,347)-(1194,380): text "左升降上下气缸Y0_7"
ellipse at (814,387)-(859,418): alarm colour if Y0_8
rectangle at (865,385)-(1194,418): text "左升降吸盘真空吸Y0_8"
ellipse at (812,426)-(857,457): alarm colour if Y0_9
rectangle at (863,424)-(1192,457): text "滚压滚轮气缸Y0_9"
ellipse at (812,464)-(857,495): alarm colour if Y0_10
rectangle at (863,462)-(1192,495): text "滚压推入气缸Y0_10"
ellipse at (812,500)-(857,531): alarm colour if Y0_11
rectangle at (863,498)-(1192,531): text "滚压下压压板气缸Y0_11"
ellipse at (812,538)-(857,569): alarm colour if Y0_12
rectangle at (863,536)-(1192,569): text "*滚压平台真空吸Y0_12"
ellipse at (812,577)-(857,608): alarm colour if Y0_13
rectangle at (863,575)-(1192,608): text "滚压翻转气缸Y0_13"
ellipse at (812,615)-(857,646): alarm colour if Y0_14
rectangle at (863,613)-(1192,646): text "右载盘真空吸Y0_14"
ellipse at (812,651)-(857,682): alarm colour if Y0_15
ellipse at (812,689)-(857,720): alarm colour if Y0_16
rectangle at (863,687)-(1192,720): text "右升降平移气缸Y0_16"
5 more shapes without text or variables
*)

(* Visualisation TC_IO3
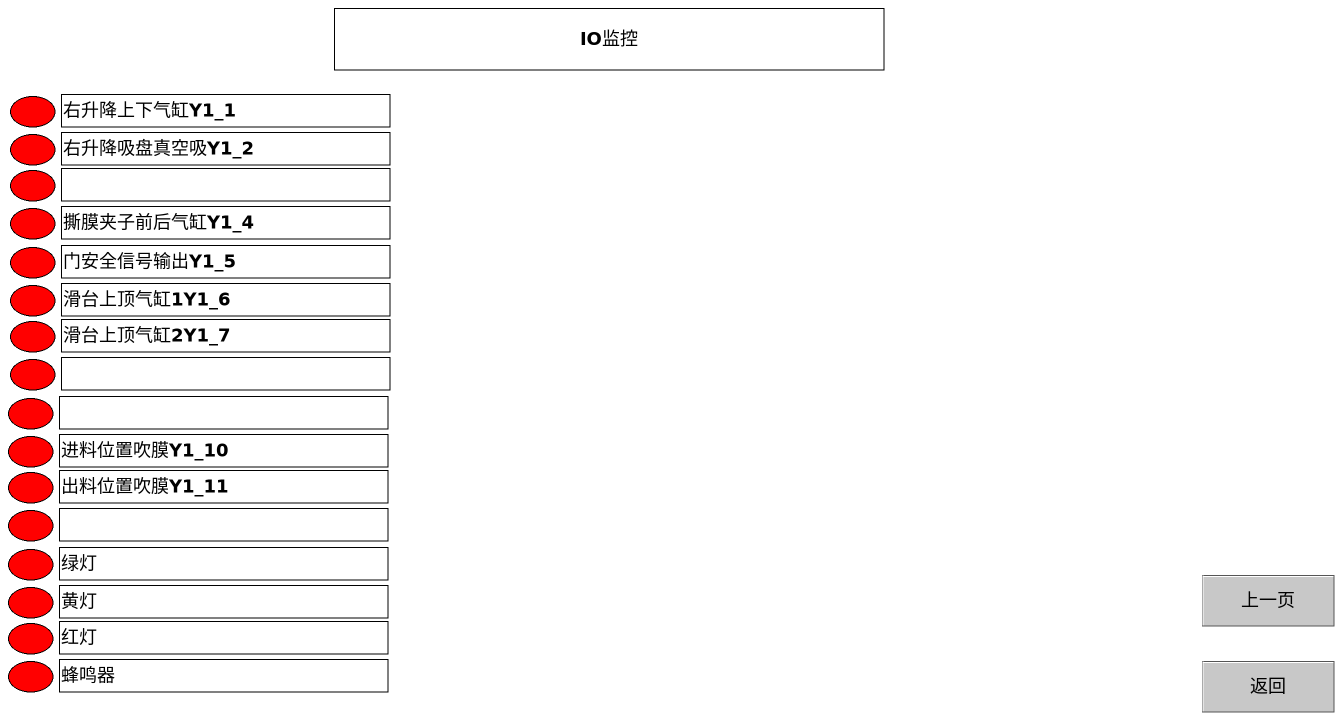
button at (1217,693)-(1349,744): text "返回"; opens TC_VIEW
button at (1217,607)-(1349,658): text "上一页"; opens TC_IO2
rounded rectangle at (349,40)-(899,102): text "IO监控"
ellipse at (25,128)-(70,159): alarm colour if Y1_1
rectangle at (76,126)-(405,159): text "右升降上下气缸Y1_1"
ellipse at (25,166)-(70,197): alarm colour if Y1_2
rectangle at (76,164)-(405,197): text "右升降吸盘真空吸Y1_2"
ellipse at (25,202)-(70,233): alarm colour if Y1_3
ellipse at (25,240)-(70,271): alarm colour if Y1_4
rectangle at (76,238)-(405,271): text "撕膜夹子前后气缸Y1_4"
ellipse at (25,279)-(70,310): alarm colour if Y1_5
rectangle at (76,277)-(405,310): text "门安全信号输出Y1_5"
ellipse at (25,317)-(70,348): alarm colour if Y1_6
rectangle at (76,315)-(405,348): text "滑台上顶气缸1Y1_6"
ellipse at (25,353)-(70,384): alarm colour if Y1_7
rectangle at (76,351)-(405,384): text "滑台上顶气缸2Y1_7"
ellipse at (25,391)-(70,422): alarm colour if Y1_8
ellipse at (23,430)-(68,461): alarm colour if Y1_9
ellipse at (23,468)-(68,499): alarm colour if Y1_10
rectangle at (74,466)-(403,499): text "进料位置吹膜Y1_10"
ellipse at (23,504)-(68,535): alarm colour if Y1_11
rectangle at (74,502)-(403,535): text "出料位置吹膜Y1_11"
ellipse at (23,542)-(68,573): alarm colour if Y1_12
ellipse at (23,581)-(68,612): alarm colour if Y1_13
rectangle at (74,579)-(403,612): text "绿灯"
ellipse at (23,619)-(68,650): alarm colour if Y1_14
rectangle at (74,617)-(403,650): text "黄灯"
ellipse at (23,655)-(68,686): alarm colour if Y1_15
rectangle at (74,653)-(403,686): text "红灯"
ellipse at (23,693)-(68,724): alarm colour if Y1_16
rectangle at (74,691)-(403,724): text "蜂鸣器"
4 more shapes without text or variables
*)

(* Visualisation TC_MESSAGE
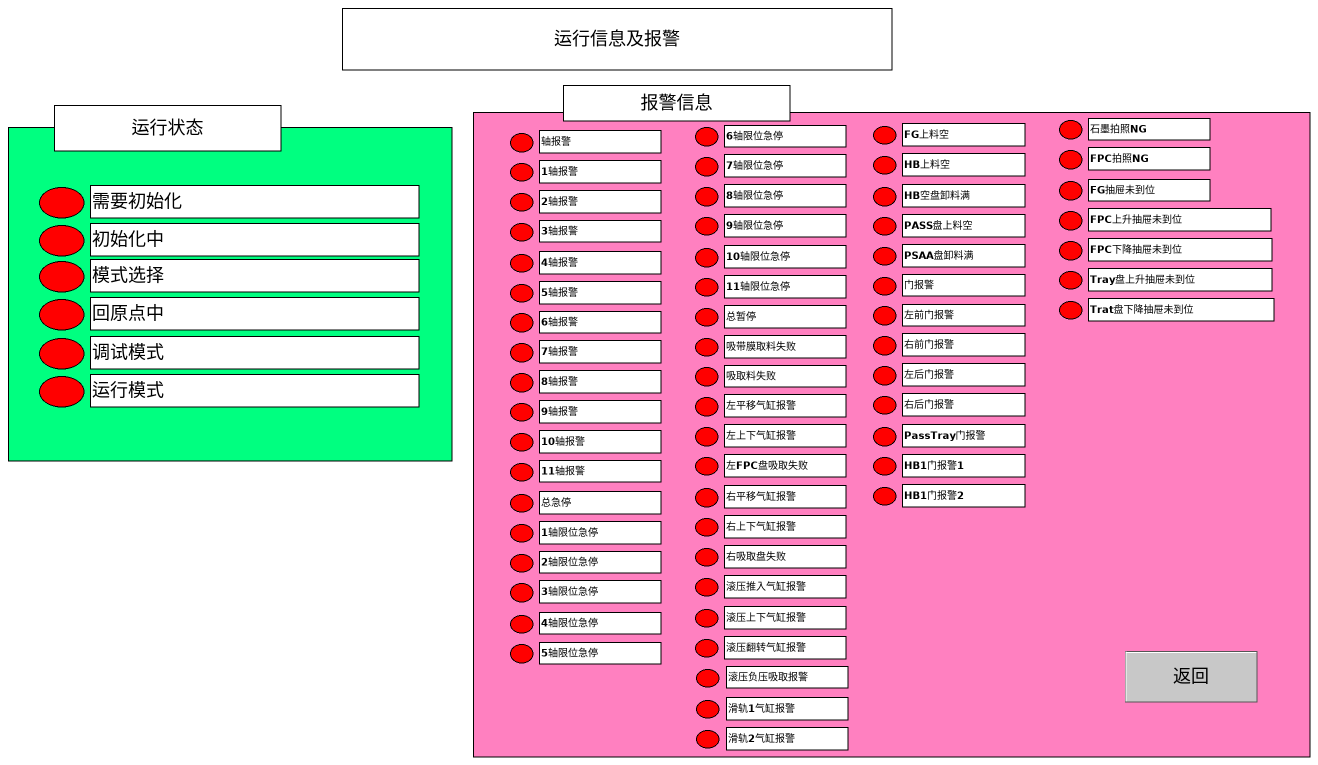
rounded rectangle at (373,7)-(923,69): text "运行信息及报警"
ellipse at (70,186)-(115,217): alarm colour if Message[0]
rectangle at (121,184)-(450,217): text "需要初始化"
ellipse at (70,224)-(115,255): alarm colour if Message[1]
rectangle at (121,222)-(450,255): text "初始化中"
ellipse at (70,260)-(115,291): alarm colour if Message[2]
rectangle at (121,258)-(450,291): text "模式选择"
ellipse at (70,298)-(115,329): alarm colour if Message[3]
rectangle at (121,296)-(450,329): text "回原点中"
ellipse at (70,337)-(115,368): alarm colour if Message[4]
rectangle at (121,335)-(450,368): text "调试模式"
ellipse at (70,375)-(115,406): alarm colour if Message[5]
rectangle at (121,373)-(450,406): text "运行模式"
rectangle at (85,104)-(312,150): text "运行状态"
button at (1156,650)-(1288,701): text "返回"; opens TC_VIEW
rectangle at (594,84)-(821,120): text "报警信息"
ellipse at (541,132)-(564,151): alarm colour if Alam[0]
rectangle at (570,129)-(692,152): text "轴报警"
ellipse at (541,162)-(564,180): alarm colour if Alam[1]
rectangle at (570,159)-(692,182): text "1轴报警"
ellipse at (541,192)-(564,210): alarm colour if Alam[2]
rectangle at (570,189)-(692,212): text "2轴报警"
ellipse at (541,222)-(564,240): alarm colour if Alam[3]
rectangle at (570,219)-(692,241): text "3轴报警"
ellipse at (541,253)-(564,271): alarm colour if Alam[04
rectangle at (570,250)-(692,273): text "4轴报警"
ellipse at (541,283)-(564,301): alarm colour if Alam[5]
rectangle at (570,280)-(692,303): text "5轴报警"
ellipse at (541,312)-(564,331): alarm colour if Alam[6]
rectangle at (570,310)-(692,332): text "6轴报警"
ellipse at (541,342)-(564,361): alarm colour if Alam[7]
rectangle at (570,339)-(692,362): text "7轴报警"
ellipse at (541,372)-(564,391): alarm colour if Alam[8]
rectangle at (570,369)-(692,392): text "8轴报警"
ellipse at (541,402)-(564,420): alarm colour if Alam[9]
rectangle at (570,399)-(692,422): text "9轴报警"
ellipse at (541,432)-(564,450): alarm colour if Alam[10]
rectangle at (570,429)-(692,452): text "10轴报警"
ellipse at (541,462)-(564,480): alarm colour if Alam[11]
rectangle at (570,459)-(692,481): text "11轴报警"
ellipse at (541,493)-(564,511): alarm colour if Alam[12]
rectangle at (570,490)-(692,513): text "总急停"
ellipse at (541,523)-(564,541): alarm colour if Alam[13]
rectangle at (570,520)-(692,543): text "1轴限位急停"
ellipse at (541,553)-(564,571): alarm colour if Alam[14]
rectangle at (570,550)-(692,572): text "2轴限位急停"
ellipse at (541,582)-(564,601): alarm colour if Alam[15]
rectangle at (570,579)-(692,602): text "3轴限位急停"
ellipse at (541,614)-(564,632): alarm colour if Alam[16]
rectangle at (570,611)-(692,633): text "4轴限位急停"
ellipse at (541,643)-(564,662): alarm colour if Alam[17]
rectangle at (570,641)-(692,663): text "5轴限位急停"
ellipse at (726,126)-(749,145): alarm colour if Alam[18]
rectangle at (755,124)-(877,146): text "6轴限位急停"
ellipse at (726,156)-(749,175): alarm colour if Alam[19]
rectangle at (755,153)-(877,176): text "7轴限位急停"
ellipse at (726,186)-(749,205): alarm colour if Alam[20]
rectangle at (755,183)-(877,206): text "8轴限位急停"
ellipse at (726,216)-(749,234): alarm colour if Alam[21]
rectangle at (755,213)-(877,236): text "9轴限位急停"
ellipse at (726,247)-(749,266): alarm colour if Alam[22]
rectangle at (755,244)-(877,267): text "10轴限位急停"
ellipse at (726,277)-(749,295): alarm colour if Alam[23]
rectangle at (755,274)-(877,297): text "11轴限位急停"
ellipse at (726,307)-(749,325): alarm colour if Alam[24]
rectangle at (755,304)-(877,327): text "总暂停"
ellipse at (726,337)-(749,355): alarm colour if Alam[25]
rectangle at (755,334)-(877,357): text "吸带膜取料失败"
ellipse at (726,366)-(749,385): alarm colour if Alam[26]
rectangle at (755,364)-(877,386): text "吸取料失败"
ellipse at (726,396)-(749,415): alarm colour if Alam[27]
rectangle at (755,393)-(877,416): text "左平移气缸报警"
ellipse at (726,426)-(749,445): alarm colour if Alam[28]
rectangle at (755,423)-(877,446): text "左上下气缸报警"
ellipse at (726,456)-(749,474): alarm colour if Alam[29]
rectangle at (755,453)-(877,476): text "左FPC盘吸取失败"
ellipse at (726,487)-(749,506): alarm colour if Alam[30]
rectangle at (755,484)-(877,507): text "右平移气缸报警"
ellipse at (726,517)-(749,535): alarm colour if Alam[31]
rectangle at (755,514)-(877,537): text "右上下气缸报警"
ellipse at (726,547)-(749,565): alarm colour if Alam[32]
rectangle at (755,544)-(877,567): text "右吸取盘失败"
ellipse at (726,577)-(749,595): alarm colour if Alam[33]
rectangle at (755,574)-(877,597): text "滚压推入气缸报警"
ellipse at (726,608)-(749,626): alarm colour if Alam[34]
rectangle at (755,605)-(877,628): text "滚压上下气缸报警"
ellipse at (726,638)-(749,656): alarm colour if Alam[35]
rectangle at (755,635)-(877,658): text "滚压翻转气缸报警"
ellipse at (904,125)-(927,143): alarm colour if Alam[39]
rectangle at (933,122)-(1056,145): text "FG上料空"
ellipse at (904,155)-(927,173): alarm colour if Alam[40]
rectangle at (933,152)-(1056,175): text "HB上料空"
ellipse at (904,186)-(927,205): alarm colour if Alam[41]
rectangle at (933,183)-(1056,206): text "HB空盘卸料满"
ellipse at (904,216)-(927,234): alarm colour if Alam[42]
rectangle at (933,213)-(1056,236): text "PASS盘上料空"
ellipse at (904,246)-(927,264): alarm colour if Alam[43]
rectangle at (933,243)-(1056,266): text "PSAA盘卸料满"
ellipse at (904,276)-(927,294): alarm colour if Alam[44]
rectangle at (933,273)-(1056,295): text "门报警"
ellipse at (904,305)-(927,324): alarm colour if Alam[45]
rectangle at (933,303)-(1056,325): text "左前门报警"
ellipse at (904,335)-(927,354): alarm colour if Alam[46]
rectangle at (933,332)-(1056,355): text "右前门报警"
ellipse at (904,365)-(927,384): alarm colour if Alam[47]
rectangle at (933,362)-(1056,385): text "左后门报警"
ellipse at (904,395)-(927,413): alarm colour if Alam[48]
rectangle at (933,392)-(1056,415): text "右后门报警"
ellipse at (904,426)-(927,445): alarm colour if Alam[49]
rectangle at (933,423)-(1056,446): text "PassTray门报警"
ellipse at (904,456)-(927,474): alarm colour if Alam[50]
rectangle at (933,453)-(1056,476): text "HB1门报警1"
ellipse at (904,486)-(927,504): alarm colour if Alam[51]
rectangle at (933,483)-(1056,506): text "HB1门报警2"
ellipse at (1090,119)-(1113,138): alarm colour if Alam[52]
rectangle at (1119,117)-(1241,139): text "石墨拍照NG"
ellipse at (1090,149)-(1113,168): alarm colour if Alam[53]
rectangle at (1119,146)-(1241,169): text "FPC拍照NG"
ellipse at (1090,180)-(1113,199): alarm colour if Alam[54]
rectangle at (1119,178)-(1241,200): text "FG抽屉未到位"
ellipse at (1090,210)-(1113,229): alarm colour if Alam[55]
rectangle at (1119,207)-(1302,230): text "FPC上升抽屉未到位"
ellipse at (1090,240)-(1113,259): alarm colour if Alam[56]
rectangle at (1119,237)-(1303,260): text "FPC下降抽屉未到位"
ellipse at (1090,270)-(1113,288): alarm colour if Alam[57]
rectangle at (1119,267)-(1303,290): text "Tray盘上升抽屉未到位"
ellipse at (1090,300)-(1113,318): alarm colour if Alam[58]
rectangle at (1119,297)-(1305,320): text "Trat盘下降抽屉未到位"
ellipse at (727,668)-(750,686): alarm colour if Alam[36]
rectangle at (757,665)-(879,687): text "滚压负压吸取报警"
ellipse at (727,699)-(750,717): alarm colour if Alam[37]
rectangle at (757,696)-(879,719): text "滑轨1气缸报警"
ellipse at (727,729)-(750,747): alarm colour if Alam[38]
rectangle at (757,726)-(879,749): text "滑轨2气缸报警"
2 more shapes without text or variables
*)

(* Visualisation TC_SPEED
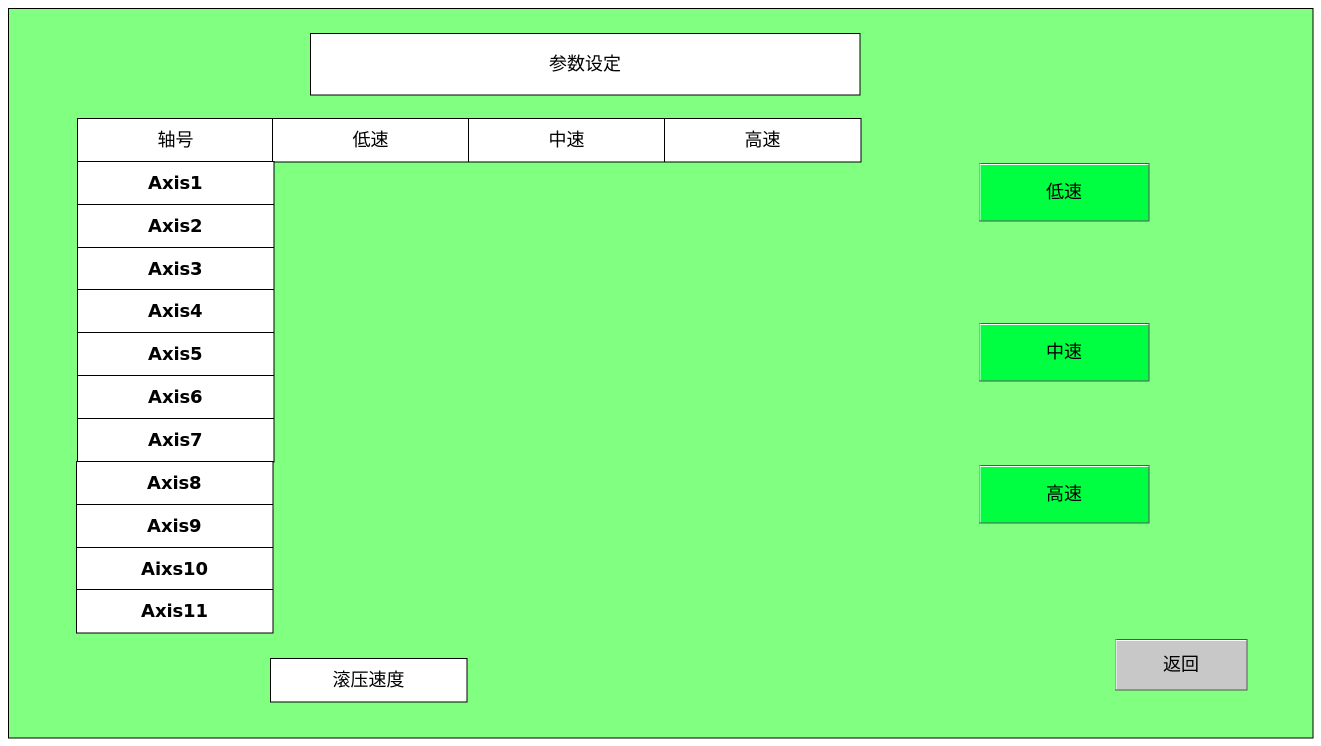
button at (1144,653)-(1276,704): text "返回"; opens TC_VIEW
rounded rectangle at (339,47)-(889,109): text "参数设定"
rectangle at (106,132)-(303,176): text "轴号"
rectangle at (301,132)-(498,176): text "低速"
rectangle at (497,132)-(694,176): text "中速"
rectangle at (693,132)-(890,176): text "高速"
button at (1008,177)-(1178,235): text "低速"; toggles M100
button at (1008,337)-(1178,395): text "中速"; toggles M101
button at (1008,479)-(1178,537): text "高速"; toggles M102
rectangle at (106,175)-(303,219): text "Axis1"
rectangle at (106,218)-(303,262): text "Axis2"
rectangle at (106,261)-(303,305): text "Axis3"
rectangle at (106,303)-(303,347): text "Axis4"
rectangle at (106,346)-(303,390): text "Axis5"
rectangle at (106,389)-(303,433): text "Axis6"
rectangle at (106,432)-(303,476): text "Axis7"
rectangle at (105,475)-(302,519): text "Axis8"
rectangle at (105,518)-(302,562): text "Axis9"
rectangle at (105,561)-(302,605): text "Aixs10"
rectangle at (105,603)-(302,647): text "Axis11"
rectangle at (299,672)-(496,716): text "滚压速度"
1 more shapes without text or variables
34 elements of other kinds (tables, trends, ...) not read
*)

(* Visualisation TC_VIEW
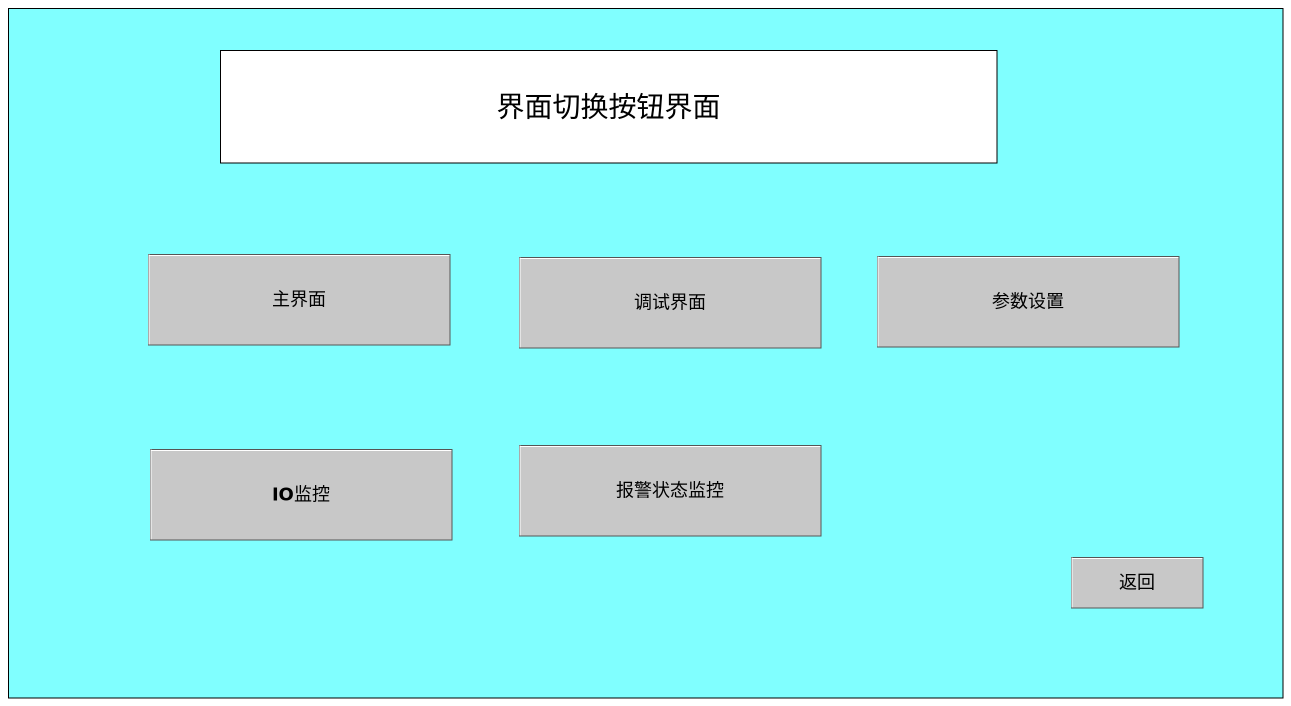
rectangle at (263,75)-(1040,188): text "界面切换按钮界面"
button at (191,279)-(493,370): text "主界面"; opens TC_HMI
button at (562,470)-(864,561): text "报警状态监控"; opens TC_MESSAGE
button at (193,474)-(495,565): text "IO监控"; opens TC_IO1
button at (562,282)-(864,373): text "调试界面"; opens TC_DEBUG
button at (920,281)-(1222,372): text "参数设置"; opens TC_SPEED
button at (1114,582)-(1246,633): text "返回"; opens TC_HMI
1 more shapes without text or variables
*)
